Yaskawa INFORM job: DPRINT3D11.JBI

/JOB
//NAME DPRINT3D11
//POS
///NPOS 944,0,0,0,0,0
///TOOL 9
///POSTYPE PULSE
///PULSE
C00000=39305,52973,-116691,73872,-117726,-90951,0
C00001=43922,55434,-109343,70072,-122046,-89427,0
C00002=34855,54702,-111321,79150,-116923,-88842,0
C00003=33073,56542,-105908,81594,-117099,-87037,0
C00004=36075,53739,-114252,77543,-116850,-89855,0
C00005=40141,50956,-123257,72181,-116164,-93028,0
C00006=40141,50893,-123279,72189,-116185,-93006,0
C00007=25718,54883,-110483,67428,-122670,-90024,0
C00008=36367,51719,-120456,76529,-115448,-91749,0
C00009=36299,54106,-112987,77479,-117287,-89472,0
C00010=40952,50916,-123219,71325,-116516,-93076,0
C00011=39945,50531,-124504,72259,-115736,-93361,0
C00012=35336,53692,-114225,78320,-116517,-89741,0
C00013=36221,54071,-113090,77546,-117224,-89494,0
C00014=35607,54392,-112113,78297,-117147,-89134,0
C00015=36480,54789,-110943,77551,-117869,-88882,0
C00016=42179,50883,-123364,69985,-116939,-93256,0
C00017=33604,54402,-112044,58649,-125681,-91811,0
C00018=34235,53812,-113837,79497,-116065,-89510,0
C00019=35137,54187,-112719,78704,-116769,-89265,0
C00020=34902,54401,-112073,79022,-116798,-89046,0
C00021=35370,54606,-111468,78618,-117176,-88914,0
C00022=35553,54440,-111967,78370,-117154,-89084,0
C00023=36112,54158,-112826,77691,-117233,-89403,0
C00024=41179,50259,-125479,70816,-115885,-93789,0
C00025=36778,53010,-116357,54404,-125157,-93511,0
C00026=39305,52913,-116713,73881,-117747,-90930,0
C00027=43892,55358,-109419,70105,-122035,-89419,0
C00028=34855,54645,-111342,79158,-116939,-88821,0
C00029=33085,56473,-105968,81585,-117112,-87030,0
C00030=36076,53681,-114273,77551,-116867,-89834,0
C00031=40141,50893,-123279,72189,-116185,-93006,0
C00032=40142,50830,-123301,72197,-116208,-92984,0
C00033=25756,54837,-110470,67404,-122722,-90001,0
C00034=36367,51658,-120476,76537,-115466,-91727,0
C00035=36299,54048,-113008,77487,-117305,-89450,0
C00036=40952,50853,-123241,71333,-116539,-93053,0
C00037=39946,50468,-124526,72267,-115759,-93339,0
C00038=35336,53633,-114246,78328,-116535,-89719,0
C00039=36221,54013,-113111,77555,-117241,-89473,0
C00040=35607,54334,-112134,78305,-117163,-89113,0
C00041=36480,54732,-110963,77560,-117886,-88861,0
C00042=42180,50820,-123386,69993,-116962,-93234,0
C00043=33604,54344,-112065,58660,-125708,-91792,0
C00044=34236,53754,-113858,79505,-116081,-89488,0
C00045=35137,54129,-112740,78712,-116785,-89244,0
C00046=34902,54343,-112094,79030,-116814,-89025,0
C00047=35370,54548,-111489,78626,-117192,-88894,0
C00048=35553,54382,-111988,78379,-117170,-89063,0
C00049=36113,54100,-112847,77699,-117251,-89382,0
C00050=41180,50194,-125500,70824,-115910,-93766,0
C00051=36764,52962,-116343,54437,-125197,-93481,0
C00052=39305,52854,-116734,73889,-117767,-90909,0
C00053=43862,55283,-109495,70139,-122024,-89410,0
C00054=34856,54587,-111363,79166,-116954,-88801,0
C00055=33098,56404,-106029,81577,-117124,-87023,0
C00056=36076,53622,-114294,77560,-116884,-89813,0
C00057=40142,50830,-123301,72197,-116208,-92984,0
C00058=40142,50767,-123323,72205,-116231,-92961,0
C00059=25794,54792,-110456,67381,-122773,-89978,0
C00060=36368,51596,-120498,76545,-115486,-91704,0
C00061=36299,53990,-113029,77496,-117322,-89430,0
C00062=40952,50790,-123263,71342,-116562,-93031,0
C00063=39946,50404,-124548,72275,-115782,-93316,0
C00064=35337,53575,-114267,78336,-116551,-89698,0
C00065=36222,53955,-113131,77563,-117258,-89452,0
C00066=35607,54276,-112155,78314,-117179,-89092,0
C00067=36480,54675,-110984,77568,-117902,-88841,0
C00068=42180,50757,-123408,70002,-116986,-93212,0
C00069=33604,54287,-112086,58672,-125736,-91774,0
C00070=34236,53695,-113879,79512,-116097,-89467,0
C00071=35137,54071,-112761,78721,-116801,-89223,0
C00072=34902,54285,-112114,79038,-116830,-89004,0
C00073=35371,54491,-111509,78635,-117208,-88873,0
C00074=35553,54325,-112009,78387,-117186,-89042,0
C00075=36113,54042,-112867,77707,-117267,-89360,0
C00076=41180,50130,-125522,70832,-115933,-93744,0
C00077=36749,52914,-116328,54470,-125238,-93452,0
C00078=39306,52794,-116755,73898,-117787,-90887,0
C00079=43832,55207,-109571,70173,-122014,-89401,0
C00080=34856,54530,-111383,79174,-116970,-88780,0
C00081=33110,56335,-106089,81568,-117137,-87016,0
C00082=36076,53564,-114315,77568,-116901,-89791,0
C00083=40142,50767,-123323,72205,-116231,-92961,0
C00084=40143,50704,-123345,72213,-116253,-92939,0
C00085=25832,54747,-110443,67357,-122825,-89955,0
C00086=36368,51535,-120519,76552,-115505,-91682,0
C00087=36300,53932,-113049,77504,-117339,-89409,0
C00088=40953,50727,-123285,71350,-116585,-93009,0
C00089=39947,50340,-124570,72283,-115805,-93293,0
C00090=35337,53516,-114288,78344,-116568,-89676,0
C00091=36222,53897,-113152,77571,-117275,-89431,0
C00092=35608,54219,-112176,78322,-117197,-89071,0
C00093=36481,54618,-111005,77577,-117919,-88820,0
C00094=42181,50693,-123430,70010,-117010,-93190,0
C00095=33605,54229,-112107,58684,-125764,-91756,0
C00096=34236,53637,-113900,79520,-116113,-89445,0
C00097=35138,54013,-112781,78729,-116819,-89201,0
C00098=34903,54228,-112135,79047,-116846,-88983,0
C00099=35371,54434,-111530,78643,-117224,-88852,0
C00100=35554,54267,-112029,78395,-117202,-89021,0
C00101=36113,53984,-112888,77716,-117284,-89340,0
C00102=41181,50066,-125544,70840,-115957,-93721,0
C00103=36735,52866,-116314,54503,-125279,-93422,0
C00104=39306,52734,-116776,73907,-117807,-90866,0
C00105=43802,55132,-109647,70206,-122004,-89393,0
C00106=34856,54473,-111404,79182,-116986,-88759,0
C00107=33122,56266,-106149,81559,-117150,-87008,0
C00108=36077,53505,-114336,77576,-116919,-89770,0
C00109=40143,50704,-123345,72213,-116253,-92939,0
C00110=40143,50641,-123365,72222,-116276,-92916,0
C00111=25870,54702,-110429,67334,-122878,-89931,0
C00112=36368,51473,-120541,76560,-115523,-91660,0
C00113=36300,53874,-113070,77513,-117356,-89388,0
C00114=40953,50664,-123307,71359,-116609,-92987,0
C00115=39947,50276,-124591,72291,-115828,-93270,0
C00116=35337,53458,-114308,78353,-116585,-89655,0
C00117=36222,53839,-113173,77580,-117292,-89410,0
C00118=35608,54161,-112196,78330,-117213,-89050,0
C00119=36481,54561,-111025,77586,-117937,-88799,0
C00120=42181,50630,-123450,70019,-117035,-93168,0
C00121=33605,54172,-112127,58695,-125791,-91738,0
C00122=34237,53579,-113920,79528,-116129,-89424,0
C00123=35138,53956,-112802,78737,-116835,-89181,0
C00124=34903,54170,-112156,79055,-116862,-88961,0
C00125=35371,54376,-111551,78651,-117240,-88831,0
C00126=35554,54210,-112050,78403,-117220,-89000,0
C00127=36114,53926,-112909,77724,-117301,-89319,0
C00128=41181,50001,-125565,70849,-115981,-93698,0
C00129=36721,52817,-116299,54537,-125320,-93393,0
C00130=39307,52675,-116797,73916,-117828,-90844,0
C00131=43772,55056,-109723,70240,-121992,-89384,0
C00132=34857,54416,-111425,79190,-117002,-88737,0
C00133=33135,56197,-106209,81551,-117162,-87001,0
C00134=36077,53447,-114357,77584,-116936,-89749,0
C00135=40143,50641,-123365,72222,-116276,-92916,0
C00136=40143,50578,-123387,72230,-116299,-92894,0
C00137=25908,54657,-110415,67310,-122930,-89908,0
C00138=36369,51412,-120561,76568,-115543,-91637,0
C00139=36300,53816,-113091,77521,-117374,-89366,0
C00140=40954,50601,-123327,71367,-116632,-92964,0
C00141=39947,50213,-124613,72299,-115851,-93247,0
C00142=35338,53399,-114329,78361,-116601,-89634,0
C00143=36223,53781,-113194,77588,-117309,-89388,0
C00144=35608,54104,-112217,78339,-117230,-89029,0
C00145=36481,54504,-111046,77594,-117953,-88778,0
C00146=42182,50567,-123472,70028,-117059,-93146,0
C00147=33605,54114,-112148,58707,-125819,-91720,0
C00148=34237,53520,-113941,79536,-116145,-89402,0
C00149=35138,53898,-112823,78745,-116851,-89159,0
C00150=34903,54113,-112176,79063,-116878,-88940,0
C00151=35372,54319,-111571,78659,-117256,-88810,0
C00152=35554,54152,-112070,78412,-117236,-88979,0
C00153=36114,53869,-112929,77733,-117318,-89297,0
C00154=41181,49937,-125587,70857,-116005,-93675,0
C00155=36707,52769,-116285,54570,-125361,-93363,0
C00156=39307,52615,-116817,73925,-117847,-90823,0
C00157=43742,54980,-109798,70274,-121982,-89376,0
C00158=34857,54358,-111445,79198,-117019,-88716,0
C00159=33147,56128,-106269,81542,-117175,-86994,0
C00160=36077,53388,-114377,77593,-116953,-89727,0
C00161=40143,50578,-123387,72230,-116299,-92894,0
C00162=40144,50515,-123408,72238,-116321,-92871,0
C00163=25945,54612,-110401,67287,-122981,-89886,0
C00164=36369,51351,-120583,76576,-115563,-91614,0
C00165=36301,53758,-113111,77530,-117391,-89345,0
C00166=40954,50538,-123349,71375,-116655,-92942,0
C00167=39948,50149,-124634,72307,-115874,-93224,0
C00168=35338,53341,-114350,78369,-116619,-89612,0
C00169=36223,53723,-113214,77597,-117326,-89367,0
C00170=35608,54046,-112237,78347,-117246,-89008,0
C00171=36482,54447,-111066,77603,-117970,-88758,0
C00172=42182,50504,-123493,70036,-117083,-93124,0
C00173=33606,54057,-112168,58719,-125846,-91701,0
C00174=34237,53462,-113962,79544,-116161,-89381,0
C00175=35139,53840,-112843,78753,-116867,-89138,0
C00176=34904,54055,-112197,79071,-116894,-88919,0
C00177=35372,54262,-111592,78668,-117272,-88789,0
C00178=35555,54095,-112091,78420,-117252,-88958,0
C00179=36114,53811,-112950,77741,-117336,-89276,0
C00180=41182,49873,-125608,70865,-116029,-93652,0
C00181=36693,52721,-116270,54603,-125402,-93334,0
C00182=39307,52556,-116838,73933,-117868,-90801,0
C00183=43712,54905,-109874,70308,-121971,-89367,0
C00184=34857,54301,-111466,79207,-117033,-88696,0
C00185=33159,56059,-106328,81533,-117189,-86986,0
C00186=36078,53330,-114398,77601,-116970,-89706,0
C00187=40144,50515,-123408,72238,-116321,-92871,0
C00188=40144,50452,-123430,72246,-116344,-92848,0
C00189=25983,54568,-110386,67264,-123034,-89862,0
C00190=36370,51289,-120604,76584,-115581,-91592,0
C00191=36301,53700,-113132,77538,-117408,-89324,0
C00192=40954,50476,-123370,71384,-116678,-92919,0
C00193=39948,50085,-124656,72315,-115897,-93201,0
C00194=35338,53283,-114370,78377,-116636,-89590,0
C00195=36223,53665,-113234,77605,-117344,-89346,0
C00196=35609,53989,-112258,78355,-117262,-88987,0
C00197=36482,54390,-111087,77612,-117986,-88737,0
C00198=42182,50441,-123515,70045,-117107,-93101,0
C00199=33606,53999,-112189,58731,-125875,-91683,0
C00200=34238,53404,-113982,79552,-116177,-89359,0
C00201=35139,53782,-112864,78762,-116884,-89117,0
C00202=34904,53998,-112217,79079,-116910,-88898,0
C00203=35372,54205,-111612,78676,-117289,-88768,0
C00204=35555,54037,-112111,78429,-117269,-88937,0
C00205=36115,53753,-112970,77749,-117352,-89255,0
C00206=41182,49809,-125630,70873,-116054,-93630,0
C00207=36679,52673,-116255,54636,-125443,-93304,0
C00208=39308,52496,-116859,73942,-117887,-90780,0
C00209=43682,54829,-109949,70342,-121960,-89358,0
C00210=34858,54244,-111486,79215,-117050,-88675,0
C00211=33172,55990,-106388,81524,-117201,-86979,0
C00212=36078,53271,-114418,77609,-116987,-89684,0
C00213=40144,50452,-123430,72246,-116344,-92848,0
C00214=40145,50389,-123450,72255,-116367,-92826,0
C00215=26021,54523,-110372,67241,-123086,-89839,0
C00216=36370,51228,-120625,76591,-115600,-91569,0
C00217=36302,53642,-113152,77547,-117425,-89302,0
C00218=40955,50413,-123391,71392,-116702,-92897,0
C00219=39949,50022,-124676,72323,-115920,-93179,0
C00220=35339,53224,-114391,78385,-116652,-89569,0
C00221=36224,53608,-113255,77614,-117361,-89325,0
C00222=35609,53931,-112278,78364,-117279,-88965,0
C00223=36482,54333,-111107,77621,-118003,-88716,0
C00224=42183,50378,-123535,70054,-117132,-93079,0
C00225=33606,53942,-112209,58743,-125903,-91665,0
C00226=34238,53346,-114003,79560,-116193,-89338,0
C00227=35139,53724,-112884,78770,-116900,-89095,0
C00228=34904,53940,-112238,79087,-116927,-88877,0
C00229=35373,54147,-111632,78685,-117306,-88747,0
C00230=35555,53980,-112132,78437,-117285,-88916,0
C00231=36115,53695,-112991,77758,-117369,-89234,0
C00232=41183,49744,-125651,70881,-116079,-93606,0
C00233=36665,52626,-116242,54670,-125483,-93274,0
C00234=39308,52436,-116879,73951,-117908,-90758,0
C00235=43651,54754,-110024,70376,-121950,-89349,0
C00236=34858,54187,-111506,79223,-117066,-88653,0
C00237=33184,55921,-106448,81516,-117214,-86972,0
C00238=36078,53213,-114439,77618,-117006,-89663,0
C00239=40145,50389,-123450,72255,-116367,-92826,0
C00240=40145,50326,-123471,72263,-116390,-92803,0
C00241=26059,54478,-110357,67218,-123139,-89816,0
C00242=36370,51166,-120645,76599,-115620,-91546,0
C00243=36302,53584,-113172,77555,-117443,-89282,0
C00244=40955,50350,-123412,71401,-116725,-92874,0
C00245=39949,49958,-124698,72331,-115943,-93155,0
C00246=35339,53166,-114411,78393,-116669,-89547,0
C00247=36224,53550,-113275,77622,-117378,-89304,0
C00248=35609,53874,-112298,78372,-117295,-88944,0
C00249=36483,54276,-111127,77629,-118021,-88695,0
C00250=42183,50315,-123556,70062,-117156,-93056,0
C00251=33607,53884,-112229,58755,-125930,-91646,0
C00252=34238,53288,-114023,79568,-116210,-89316,0
C00253=35140,53667,-112904,78778,-116916,-89074,0
C00254=34905,53883,-112258,79096,-116943,-88856,0
C00255=35373,54090,-111653,78693,-117322,-88726,0
C00256=35556,53923,-112152,78445,-117301,-88895,0
C00257=36115,53637,-113011,77766,-117386,-89213,0
C00258=41183,49680,-125673,70890,-116103,-93584,0
C00259=36650,52578,-116227,54703,-125525,-93245,0
C00260=39308,52377,-116900,73960,-117929,-90737,0
C00261=43621,54678,-110099,70410,-121939,-89340,0
C00262=34858,54130,-111527,79232,-117082,-88632,0
C00263=33197,55852,-106507,81507,-117227,-86964,0
C00264=36079,53155,-114459,77626,-117023,-89641,0
C00265=40145,50326,-123471,72263,-116390,-92803,0
C00266=40145,50263,-123493,72271,-116413,-92781,0
C00267=26097,54434,-110343,67195,-123191,-89793,0
C00268=36371,51105,-120666,76607,-115638,-91524,0
C00269=36302,53527,-113193,77564,-117460,-89260,0
C00270=40956,50287,-123433,71409,-116748,-92851,0
C00271=39949,49894,-124719,72339,-115966,-93133,0
C00272=35339,53107,-114431,78402,-116686,-89526,0
C00273=36224,53492,-113295,77631,-117395,-89282,0
C00274=35610,53816,-112318,78381,-117313,-88923,0
C00275=36483,54219,-111147,77638,-118038,-88674,0
C00276=42184,50252,-123578,70071,-117181,-93034,0
C00277=33607,53827,-112249,58767,-125959,-91628,0
C00278=34239,53229,-114043,79575,-116226,-89294,0
C00279=35140,53609,-112925,78786,-116933,-89053,0
C00280=34905,53825,-112278,79104,-116959,-88834,0
C00281=35373,54033,-111673,78702,-117338,-88705,0
C00282=35556,53865,-112172,78454,-117318,-88874,0
C00283=36116,53580,-113031,77775,-117403,-89192,0
C00284=41184,49616,-125693,70898,-116127,-93560,0
C00285=36636,52530,-116212,54736,-125565,-93215,0
C00286=39309,52317,-116921,73969,-117948,-90715,0
C00287=43591,54602,-110174,70444,-121929,-89331,0
C00288=34859,54073,-111547,79240,-117098,-88611,0
C00289=33209,55783,-106566,81498,-117240,-86956,0
C00290=36079,53096,-114480,77635,-117040,-89620,0
C00291=40145,50263,-123493,72271,-116413,-92781,0
C00292=40146,50200,-123514,72280,-116436,-92757,0
C00293=26135,54389,-110328,67172,-123243,-89770,0
C00294=36371,51043,-120687,76615,-115658,-91501,0
C00295=36303,53469,-113213,77572,-117477,-89239,0
C00296=40956,50224,-123454,71418,-116773,-92829,0
C00297=39950,49831,-124740,72348,-115989,-93110,0
C00298=35340,53049,-114451,78410,-116704,-89504,0
C00299=36225,53434,-113315,77639,-117413,-89261,0
C00300=35610,53759,-112338,78389,-117329,-88901,0
C00301=36483,54162,-111167,77647,-118054,-88653,0
C00302=42184,50189,-123599,70080,-117205,-93012,0
C00303=33607,53769,-112269,58779,-125987,-91610,0
C00304=34239,53171,-114063,79584,-116242,-89273,0
C00305=35140,53551,-112945,78795,-116950,-89031,0
C00306=34905,53768,-112298,79112,-116975,-88813,0
C00307=35374,53976,-111693,78710,-117354,-88683,0
C00308=35556,53808,-112192,78462,-117335,-88852,0
C00309=36116,53522,-113051,77784,-117421,-89170,0
C00310=41184,49552,-125714,70906,-116151,-93537,0
C00311=36622,52482,-116196,54770,-125606,-93185,0
C00312=39309,52258,-116940,73978,-117969,-90694,0
C00313=43561,54527,-110249,70478,-121919,-89322,0
C00314=34859,54015,-111567,79248,-117114,-88590,0
C00315=33222,55714,-106626,81490,-117253,-86949,0
C00316=36079,53038,-114500,77643,-117058,-89598,0
C00317=40146,50200,-123514,72280,-116436,-92757,0
C00318=40146,50137,-123534,72288,-116458,-92735,0
C00319=26173,54345,-110313,67149,-123295,-89746,0
C00320=36371,50982,-120707,76623,-115677,-91478,0
C00321=36303,53411,-113233,77581,-117494,-89218,0
C00322=40956,50161,-123474,71427,-116796,-92806,0
C00323=39950,49767,-124762,72356,-116012,-93086,0
C00324=35340,52991,-114472,78418,-116720,-89482,0
C00325=36225,53376,-113336,77648,-117430,-89239,0
C00326=35611,53701,-112358,78398,-117346,-88881,0
C00327=36484,54105,-111187,77656,-118071,-88632,0
C00328=42184,50126,-123619,70089,-117229,-92989,0
C00329=33608,53712,-112289,58790,-126014,-91591,0
C00330=34239,53113,-114083,79591,-116258,-89251,0
C00331=35141,53494,-112965,78803,-116966,-89010,0
C00332=34906,53710,-112318,79121,-116991,-88792,0
C00333=35374,53919,-111713,78718,-117370,-88662,0
C00334=35556,53750,-112212,78471,-117352,-88831,0
C00335=36116,53464,-113071,77792,-117438,-89149,0
C00336=41184,49487,-125736,70915,-116175,-93515,0
C00337=36608,52435,-116181,54804,-125646,-93155,0
C00338=39310,52199,-116961,73987,-117988,-90672,0
C00339=43530,54451,-110324,70512,-121908,-89313,0
C00340=34859,53958,-111587,79257,-117130,-88569,0
C00341=33234,55645,-106685,81481,-117267,-86941,0
C00342=36080,52979,-114520,77652,-117075,-89576,0
C00343=40146,50137,-123534,72288,-116458,-92735,0
C00344=40147,50074,-123555,72297,-116481,-92712,0
C00345=26210,54300,-110298,67126,-123348,-89723,0
C00346=36372,50921,-120728,76631,-115697,-91455,0
C00347=36303,53353,-113253,77590,-117511,-89196,0
C00348=40957,50098,-123495,71435,-116819,-92783,0
C00349=39951,49704,-124782,72364,-116035,-93063,0
C00350=35340,52932,-114492,78427,-116737,-89461,0
C00351=36225,53318,-113355,77657,-117447,-89218,0
C00352=35611,53644,-112378,78406,-117362,-88859,0
C00353=36484,54048,-111207,77665,-118088,-88611,0
C00354=42185,50063,-123640,70098,-117253,-92967,0
C00355=33608,53655,-112309,58803,-126043,-91572,0
C00356=34239,53055,-114103,79599,-116274,-89229,0
C00357=35141,53436,-112985,78811,-116983,-88989,0
C00358=34906,53653,-112338,79129,-117007,-88770,0
C00359=35374,53862,-111733,78727,-117387,-88641,0
C00360=35557,53693,-112232,78480,-117368,-88810,0
C00361=36117,53406,-113091,77801,-117455,-89127,0
C00362=41185,49423,-125757,70923,-116199,-93491,0
C00363=36594,52387,-116166,54837,-125688,-93126,0
C00364=39310,52139,-116981,73996,-118009,-90650,0
C00365=43500,54376,-110398,70546,-121898,-89304,0
C00366=34860,53901,-111607,79265,-117146,-88548,0
C00367=33247,55577,-106744,81473,-117279,-86934,0
C00368=36080,52921,-114540,77660,-117093,-89555,0
C00369=40147,50074,-123555,72297,-116481,-92712,0
C00370=40147,50011,-123576,72305,-116504,-92689,0
C00371=26248,54256,-110282,67104,-123401,-89700,0
C00372=36372,50859,-120748,76639,-115717,-91433,0
C00373=36304,53296,-113273,77598,-117529,-89175,0
C00374=40957,50035,-123516,71444,-116843,-92761,0
C00375=39951,49640,-124803,72372,-116058,-93040,0
C00376=35341,52874,-114512,78435,-116754,-89439,0
C00377=36226,53260,-113375,77665,-117464,-89196,0
C00378=35611,53587,-112398,78415,-117379,-88838,0
C00379=36484,53991,-111227,77674,-118106,-88590,0
C00380=42185,50000,-123661,70106,-117278,-92944,0
C00381=33608,53597,-112329,58815,-126070,-91554,0
C00382=34240,52997,-114123,79608,-116290,-89207,0
C00383=35141,53378,-113004,78820,-116999,-88967,0
C00384=34906,53596,-112358,79137,-117023,-88749,0
C00385=35375,53805,-111753,78736,-117403,-88620,0
C00386=35557,53636,-112252,78488,-117385,-88788,0
C00387=36117,53349,-113111,77809,-117472,-89106,0
C00388=41185,49359,-125777,70931,-116224,-93468,0
C00389=36580,52340,-116151,54871,-125728,-93096,0
C00390=39310,52080,-117001,74006,-118030,-90628,0
C00391=43470,54300,-110472,70580,-121887,-89295,0
C00392=34860,53844,-111626,79273,-117162,-88526,0
C00393=33259,55508,-106803,81464,-117292,-86926,0
C00394=36080,52863,-114560,77669,-117110,-89533,0
C00395=40147,50011,-123576,72305,-116504,-92689,0
C00396=40147,49948,-123596,72314,-116527,-92666,0
C00397=26286,54212,-110267,67081,-123454,-89677,0
C00398=36372,50798,-120768,76647,-115736,-91409,0
C00399=36304,53238,-113292,77607,-117546,-89153,0
C00400=40958,49973,-123537,71453,-116866,-92738,0
C00401=39951,49576,-124824,72381,-116081,-93017,0
C00402=35341,52816,-114531,78443,-116771,-89417,0
C00403=36226,53203,-113395,77674,-117482,-89175,0
C00404=35611,53529,-112418,78424,-117395,-88816,0
C00405=36485,53934,-111247,77682,-118122,-88569,0
C00406=42186,49938,-123681,70115,-117302,-92922,0
C00407=33608,53540,-112349,58827,-126098,-91535,0
C00408=34240,52939,-114143,79616,-116306,-89186,0
C00409=35142,53321,-113024,78828,-117016,-88946,0
C00410=34907,53538,-112378,79146,-117039,-88727,0
C00411=35375,53747,-111772,78744,-117420,-88599,0
C00412=35557,53579,-112272,78497,-117401,-88767,0
C00413=36117,53291,-113131,77818,-117490,-89084,0
C00414=41186,49295,-125798,70940,-116249,-93445,0
C00415=36566,52292,-116135,54904,-125769,-93066,0
C00416=39311,52020,-117021,74015,-118050,-90607,0
C00417=43439,54224,-110547,70615,-121877,-89286,0
C00418=34860,53787,-111646,79282,-117178,-88505,0
C00419=33272,55439,-106862,81455,-117306,-86918,0
C00420=36081,52805,-114580,77677,-117128,-89511,0
C00421=40147,49948,-123596,72314,-116527,-92666,0
C00422=40148,49886,-123617,72322,-116550,-92643,0
C00423=26324,54168,-110251,67059,-123507,-89654,0
C00424=36373,50737,-120788,76655,-115754,-91387,0
C00425=36304,53180,-113312,77616,-117563,-89132,0
C00426=40958,49910,-123557,71461,-116890,-92715,0
C00427=39952,49513,-124844,72389,-116105,-92994,0
C00428=35341,52758,-114551,78452,-116789,-89395,0
C00429=36226,53145,-113415,77683,-117500,-89153,0
C00430=35612,53472,-112438,78432,-117413,-88795,0
C00431=36485,53877,-111266,77691,-118139,-88548,0
C00432=42186,49875,-123702,70124,-117326,-92899,0
C00433=33609,53483,-112369,58839,-126127,-91517,0
C00434=34241,52881,-114163,79624,-116322,-89164,0
C00435=35142,53263,-113044,78837,-117032,-88924,0
C00436=34907,53481,-112397,79154,-117056,-88706,0
C00437=35375,53690,-111792,78753,-117436,-88577,0
C00438=35558,53521,-112291,78505,-117418,-88745,0
C00439=36118,53233,-113151,77827,-117507,-89063,0
C00440=41186,49231,-125819,70948,-116273,-93422,0
C00441=36552,52245,-116120,54938,-125810,-93036,0
C00442=39311,51961,-117041,74024,-118070,-90585,0
C00443=43409,54149,-110621,70649,-121867,-89276,0
C00444=34861,53730,-111666,79290,-117194,-88484,0
C00445=33284,55370,-106921,81447,-117320,-86911,0
C00446=36081,52746,-114599,77686,-117145,-89490,0
C00447=40148,49886,-123617,72322,-116550,-92643,0
C00448=40148,49823,-123636,72331,-116573,-92620,0
C00449=26361,54124,-110236,67037,-123560,-89630,0
C00450=36373,50676,-120808,76663,-115774,-91364,0
C00451=36304,53122,-113332,77625,-117580,-89110,0
C00452=40958,49847,-123577,71470,-116913,-92692,0
C00453=39952,49449,-124864,72398,-116128,-92970,0
C00454=35342,52699,-114571,78460,-116805,-89374,0
C00455=36227,53087,-113435,77692,-117517,-89132,0
C00456=35612,53415,-112457,78441,-117429,-88774,0
C00457=36485,53821,-111286,77700,-118156,-88527,0
C00458=42187,49812,-123722,70133,-117351,-92876,0
C00459=33609,53425,-112388,58851,-126154,-91498,0
C00460=34241,52823,-114183,79632,-116338,-89142,0
C00461=35142,53206,-113064,78845,-117048,-88903,0
C00462=34907,53424,-112417,79163,-117073,-88684,0
C00463=35376,53633,-111811,78761,-117453,-88556,0
C00464=35558,53464,-112311,78514,-117435,-88725,0
C00465=36118,53176,-113170,77836,-117524,-89041,0
C00466=41187,49167,-125839,70957,-116298,-93399,0
C00467=36538,52197,-116104,54972,-125850,-93006,0
C00468=39311,51901,-117061,74033,-118091,-90563,0
C00469=43378,54073,-110695,70684,-121856,-89267,0
C00470=34861,53673,-111685,79299,-117210,-88462,0
C00471=33296,55301,-106979,81438,-117332,-86902,0
C00472=36081,52688,-114619,77694,-117163,-89468,0
C00473=40148,49823,-123636,72331,-116573,-92620,0
C00474=40149,49760,-123657,72340,-116596,-92597,0
C00475=26399,54080,-110220,67014,-123612,-89607,0
C00476=36374,50614,-120828,76672,-115794,-91341,0
C00477=36305,53065,-113351,77633,-117598,-89089,0
C00478=40959,49784,-123597,71479,-116937,-92670,0
C00479=39953,49386,-124884,72406,-116151,-92947,0
C00480=35342,52641,-114590,78468,-116822,-89352,0
C00481=36227,53029,-113454,77700,-117534,-89110,0
C00482=35612,53357,-112477,78449,-117446,-88752,0
C00483=36486,53764,-111305,77709,-118173,-88506,0
C00484=42187,49749,-123742,70142,-117376,-92854,0
C00485=33609,53368,-112408,58863,-126183,-91480,0
C00486=34241,52764,-114202,79640,-116354,-89120,0
C00487=35143,53148,-113083,78853,-117066,-88881,0
C00488=34908,53366,-112436,79171,-117089,-88663,0
C00489=35376,53576,-111831,78770,-117469,-88535,0
C00490=35558,53407,-112330,78522,-117452,-88703,0
C00491=36118,53118,-113190,77844,-117541,-89020,0
C00492=41187,49103,-125860,70965,-116322,-93375,0
C00493=36524,52150,-116089,55005,-125891,-92976,0
C00494=39312,51842,-117081,74042,-118111,-90541,0
C00495=43348,53998,-110769,70718,-121846,-89258,0
C00496=34861,53616,-111705,79307,-117227,-88441,0
C00497=33309,55232,-107038,81430,-117346,-86895,0
C00498=36082,52630,-114639,77703,-117181,-89446,0
C00499=40149,49760,-123657,72340,-116596,-92597,0
C00500=40149,49697,-123677,72348,-116619,-92574,0
C00501=26437,54036,-110204,66992,-123665,-89584,0
C00502=36374,50553,-120849,76680,-115813,-91318,0
C00503=36305,53007,-113371,77642,-117616,-89067,0
C00504=40959,49721,-123618,71488,-116960,-92647,0
C00505=39953,49322,-124905,72414,-116174,-92924,0
C00506=35342,52583,-114610,78477,-116839,-89330,0
C00507=36227,52972,-113474,77709,-117552,-89089,0
C00508=35613,53300,-112496,78458,-117463,-88731,0
C00509=36486,53707,-111325,77718,-118191,-88484,0
C00510=42187,49686,-123763,70151,-117400,-92831,0
C00511=33610,53311,-112427,58875,-126211,-91460,0
C00512=34241,52706,-114222,79648,-116372,-89098,0
C00513=35143,53091,-113103,78862,-117082,-88859,0
C00514=34908,53309,-112456,79179,-117105,-88642,0
C00515=35376,53519,-111850,78779,-117485,-88513,0
C00516=35559,53350,-112350,78531,-117468,-88682,0
C00517=36119,53061,-113209,77853,-117559,-88998,0
C00518=41187,49038,-125881,70974,-116346,-93352,0
C00519=36510,52103,-116073,55039,-125931,-92946,0
C00520=39312,51783,-117100,74051,-118132,-90519,0
C00521=43318,53922,-110842,70753,-121836,-89248,0
C00522=34861,53559,-111724,79316,-117243,-88419,0
C00523=33322,55163,-107097,81421,-117359,-86887,0
C00524=36082,52571,-114658,77712,-117198,-89424,0
C00525=40149,49697,-123677,72348,-116619,-92574,0
C00526=40149,49634,-123697,72357,-116642,-92551,0
C00527=26474,53992,-110188,66970,-123718,-89561,0
C00528=36374,50492,-120868,76688,-115833,-91295,0
C00529=36306,52950,-113390,77651,-117633,-89045,0
C00530=40960,49659,-123638,71497,-116984,-92624,0
C00531=39954,49259,-124925,72423,-116198,-92901,0
C00532=35343,52525,-114629,78485,-116856,-89308,0
C00533=36228,52914,-113493,77718,-117569,-89067,0
C00534=35613,53243,-112516,78467,-117479,-88709,0
C00535=36486,53650,-111344,77727,-118207,-88463,0
C00536=42188,49623,-123782,70160,-117425,-92808,0
C00537=33610,53254,-112446,58888,-126239,-91442,0
C00538=34242,52648,-114241,79656,-116388,-89076,0
C00539=35143,53033,-113122,78871,-117099,-88838,0
C00540=34908,53252,-112475,79188,-117121,-88620,0
C00541=35377,53462,-111870,78787,-117502,-88492,0
C00542=35559,53292,-112369,78540,-117485,-88660,0
C00543=36119,53003,-113229,77862,-117576,-88977,0
C00544=41188,48974,-125900,70982,-116372,-93328,0
C00545=36496,52056,-116057,55073,-125973,-92916,0
C00546=39312,51723,-117120,74061,-118152,-90498,0
C00547=43287,53847,-110916,70787,-121827,-89239,0
C00548=34862,53502,-111744,79324,-117259,-88398,0
C00549=33334,55094,-107155,81413,-117372,-86879,0
C00550=36082,52513,-114678,77720,-117216,-89403,0
C00551=40149,49634,-123697,72357,-116642,-92551,0
C00552=40150,49572,-123717,72366,-116665,-92528,0
C00553=26512,53948,-110172,66948,-123771,-89537,0
C00554=36375,50431,-120888,76696,-115852,-91272,0
C00555=36306,52892,-113409,77660,-117651,-89024,0
C00556=40960,49596,-123658,71506,-117007,-92601,0
C00557=39954,49195,-124945,72432,-116221,-92877,0
C00558=35343,52467,-114649,78494,-116874,-89286,0
C00559=36228,52856,-113512,77727,-117586,-89045,0
C00560=35613,53185,-112535,78475,-117497,-88687,0
C00561=36487,53593,-111363,77736,-118224,-88442,0
C00562=42188,49560,-123802,70170,-117449,-92785,0
C00563=33610,53196,-112466,58900,-126268,-91423,0
C00564=34242,52590,-114260,79665,-116404,-89054,0
C00565=35144,52976,-113141,78879,-117115,-88816,0
C00566=34909,53195,-112494,79197,-117137,-88599,0
C00567=35377,53405,-111889,78796,-117518,-88470,0
C00568=35559,53235,-112388,78549,-117501,-88638,0
C00569=36119,52946,-113248,77871,-117593,-88955,0
C00570=41188,48910,-125921,70991,-116396,-93305,0
C00571=36482,52008,-116041,55107,-126013,-92886,0
C00572=39313,51664,-117139,74070,-118172,-90476,0
C00573=43257,53771,-110990,70822,-121816,-89229,0
C00574=34862,53445,-111763,79333,-117275,-88376,0
C00575=33347,55025,-107213,81404,-117386,-86871,0
C00576=36083,52455,-114697,77729,-117233,-89381,0
C00577=40150,49572,-123717,72366,-116665,-92528,0
C00578=40150,49509,-123738,72375,-116688,-92505,0
C00579=26549,53905,-110155,66926,-123824,-89514,0
C00580=36375,50369,-120907,76704,-115872,-91249,0
C00581=36306,52834,-113429,77669,-117668,-89002,0
C00582=40961,49533,-123678,71514,-117031,-92578,0
C00583=39954,49132,-124965,72440,-116244,-92854,0
C00584=35343,52408,-114668,78502,-116891,-89264,0
C00585=36228,52799,-113532,77735,-117603,-89024,0
C00586=35614,53128,-112554,78484,-117513,-88666,0
C00587=36487,53537,-111382,77746,-118241,-88420,0
C00588=42189,49498,-123823,70179,-117474,-92763,0
C00589=33611,53139,-112485,58912,-126296,-91404,0
C00590=34242,52532,-114280,79673,-116420,-89032,0
C00591=35144,52918,-113160,78888,-117132,-88794,0
C00592=34909,53138,-112514,79205,-117154,-88577,0
C00593=35377,53348,-111908,78805,-117536,-88449,0
C00594=35560,53178,-112408,78557,-117518,-88617,0
C00595=36120,52888,-113267,77880,-117610,-88933,0
C00596=41189,48846,-125942,71000,-116420,-93282,0
C00597=36468,51961,-116024,55141,-126053,-92855,0
C00598=39313,51605,-117159,74079,-118193,-90454,0
C00599=43226,53695,-111063,70857,-121806,-89219,0
C00600=34862,53388,-111782,79341,-117291,-88355,0
C00601=33359,54956,-107271,81396,-117400,-86863,0
C00602=36083,52397,-114716,77738,-117251,-89359,0
C00603=40150,49509,-123738,72375,-116688,-92505,0
C00604=40151,49446,-123757,72383,-116712,-92482,0
C00605=26587,53861,-110139,66905,-123878,-89490,0
C00606=36375,50308,-120927,76713,-115891,-91225,0
C00607=36307,52777,-113448,77678,-117685,-88980,0
C00608=40961,49470,-123697,71523,-117055,-92555,0
C00609=39955,49068,-124986,72449,-116268,-92830,0
C00610=35344,52350,-114687,78511,-116908,-89242,0
C00611=36229,52741,-113551,77744,-117622,-89002,0
C00612=35614,53071,-112573,78493,-117530,-88644,0
C00613=36487,53480,-111402,77755,-118258,-88399,0
C00614=42189,49435,-123842,70188,-117499,-92740,0
C00615=33611,53082,-112504,58925,-126324,-91386,0
C00616=34243,52474,-114299,79681,-116436,-89010,0
C00617=35144,52861,-113180,78896,-117148,-88772,0
C00618=34909,53080,-112533,79214,-117170,-88555,0
C00619=35378,53291,-111927,78813,-117552,-88427,0
C00620=35560,53121,-112427,78566,-117534,-88595,0
C00621=36120,52830,-113286,77888,-117628,-88912,0
C00622=41189,48782,-125961,71008,-116445,-93258,0
C00623=36454,51914,-116008,55175,-126095,-92825,0
C00624=39314,51545,-117178,74088,-118214,-90432,0
C00625=43195,53620,-111136,70892,-121796,-89209,0
C00626=34863,53332,-111801,79350,-117307,-88333,0
C00627=33372,54887,-107330,81388,-117413,-86855,0
C00628=36083,52339,-114736,77746,-117269,-89337,0
C00629=40151,49446,-123757,72383,-116712,-92482,0
C00630=40151,49383,-123777,72392,-116735,-92459,0
C00631=26624,53817,-110122,66883,-123931,-89467,0
C00632=36376,50247,-120946,76721,-115911,-91202,0
C00633=36307,52719,-113467,77686,-117703,-88959,0
C00634=40961,49408,-123717,71532,-117078,-92532,0
C00635=39955,49005,-125005,72457,-116291,-92807,0
C00636=35344,52292,-114706,78519,-116925,-89220,0
C00637=36229,52684,-113570,77753,-117639,-88980,0
C00638=35614,53014,-112592,78502,-117547,-88623,0
C00639=36488,53423,-111421,77764,-118276,-88378,0
C00640=42190,49372,-123862,70197,-117523,-92717,0
C00641=33611,53025,-112523,58937,-126353,-91367,0
C00642=34243,52417,-114318,79689,-116453,-88988,0
C00643=35145,52803,-113199,78905,-117166,-88751,0
C00644=34909,53023,-112552,79222,-117186,-88534,0
C00645=35378,53235,-111946,78822,-117568,-88406,0
C00646=35560,53064,-112446,78575,-117552,-88574,0
C00647=36120,52773,-113305,77897,-117645,-88890,0
C00648=41190,48718,-125981,71017,-116469,-93235,0
C00649=36440,51867,-115991,55209,-126135,-92795,0
C00650=39314,51486,-117198,74098,-118234,-90410,0
C00651=43165,53544,-111209,70926,-121786,-89200,0
C00652=34863,53275,-111820,79359,-117323,-88312,0
C00653=33384,54818,-107388,81379,-117426,-86847,0
C00654=36084,52281,-114755,77755,-117286,-89315,0
C00655=40151,49383,-123777,72392,-116735,-92459,0
C00656=40151,49321,-123796,72401,-116758,-92435,0
C00657=26662,53774,-110105,66861,-123984,-89443,0
C00658=36376,50186,-120966,76729,-115930,-91179,0
C00659=36307,52662,-113486,77695,-117721,-88937,0
C00660=40962,49345,-123738,71541,-117102,-92508,0
C00661=39956,48941,-125025,72466,-116314,-92783,0
C00662=35344,52234,-114725,78528,-116943,-89198,0
C00663=36229,52626,-113589,77762,-117656,-88958,0
C00664=35615,52957,-112611,78511,-117563,-88601,0
C00665=36488,53367,-111439,77773,-118293,-88357,0
C00666=42190,49309,-123882,70206,-117548,-92694,0
C00667=33612,52968,-112542,58950,-126381,-91348,0
C00668=34243,52359,-114337,79698,-116469,-88966,0
C00669=35145,52746,-113218,78914,-117182,-88729,0
C00670=34910,52966,-112571,79231,-117202,-88512,0
C00671=35378,53178,-111965,78831,-117585,-88384,0
C00672=35561,53007,-112465,78584,-117569,-88552,0
C00673=36121,52716,-113324,77906,-117662,-88868,0
C00674=41190,48654,-126001,71026,-116494,-93211,0
C00675=36426,51821,-115975,55243,-126175,-92765,0
C00676=39314,51427,-117216,74107,-118255,-90388,0
C00677=43134,53469,-111282,70961,-121776,-89190,0
C00678=34863,53218,-111839,79367,-117339,-88290,0
C00679=33397,54749,-107445,81371,-117440,-86839,0
C00680=36084,52223,-114774,77764,-117305,-89293,0
C00681=40151,49321,-123796,72401,-116758,-92435,0
C00682=40152,49258,-123816,72410,-116781,-92412,0
C00683=26699,53731,-110088,66840,-124038,-89420,0
C00684=36376,50125,-120985,76738,-115950,-91156,0
C00685=36308,52604,-113505,77704,-117738,-88915,0
C00686=40962,49282,-123757,71550,-117127,-92486,0
C00687=39956,48878,-125045,72474,-116338,-92760,0
C00688=35344,52176,-114744,78537,-116960,-89175,0
C00689=36230,52568,-113608,77771,-117674,-88937,0
C00690=35615,52900,-112630,78520,-117580,-88579,0
C00691=36488,53310,-111458,77782,-118310,-88335,0
C00692=42190,49246,-123902,70215,-117572,-92671,0
C00693=39823,48305,-126937,72401,-115720,-93319,0
C00694=34244,52301,-114356,79706,-116485,-88944,0
C00695=35145,52688,-113237,78922,-117199,-88707,0
C00696=34910,52909,-112590,79240,-117220,-88490,0
C00697=35378,53121,-111984,78840,-117601,-88362,0
C00698=35561,52950,-112484,78593,-117585,-88530,0
C00699=36121,52658,-113343,77915,-117680,-88846,0
C00700=41190,48590,-126021,71034,-116519,-93188,0
C00701=36412,51774,-115959,55277,-126216,-92735,0
C00702=39315,51368,-117236,74117,-118275,-90366,0
C00703=43103,53393,-111355,70996,-121766,-89179,0
C00704=34864,53161,-111858,79376,-117355,-88268,0
C00705=33409,54680,-107503,81362,-117454,-86831,0
C00706=36084,52165,-114793,77773,-117322,-89271,0
C00707=40152,49258,-123816,72410,-116781,-92412,0
C00708=40152,49195,-123835,72419,-116804,-92389,0
C00709=26737,53687,-110071,66818,-124090,-89397,0
C00710=36377,50064,-121005,76746,-115969,-91133,0
C00711=36308,52547,-113524,77713,-117756,-88893,0
C00712=40963,49220,-123777,71559,-117150,-92463,0
C00713=39956,48814,-125065,72483,-116361,-92736,0
C00714=35345,52118,-114763,78545,-116977,-89153,0
C00715=36230,52511,-113626,77780,-117692,-88915,0
C00716=35615,52842,-112649,78528,-117598,-88558,0
C00717=36489,53253,-111477,77791,-118327,-88314,0
C00718=42191,49184,-123921,70225,-117598,-92648,0
C00719=39823,48241,-126956,72410,-115744,-93295,0
C00720=34244,52243,-114375,79714,-116501,-88922,0
C00721=35146,52631,-113255,78931,-117215,-88685,0
C00722=34911,52852,-112608,79248,-117236,-88468,0
C00723=35379,53064,-112003,78849,-117618,-88341,0
C00724=35561,52893,-112502,78601,-117602,-88509,0
C00725=36121,52601,-113362,77924,-117698,-88825,0
C00726=41191,48526,-126041,71043,-116544,-93164,0
C00727=36398,51727,-115942,55311,-126257,-92705,0
C00728=39315,51308,-117255,74126,-118295,-90343,0
C00729=43073,53318,-111428,71031,-121756,-89170,0
C00730=34864,53104,-111877,79385,-117371,-88247,0
C00731=33422,54611,-107561,81354,-117468,-86822,0
C00732=36085,52106,-114812,77782,-117339,-89248,0
C00733=40152,49195,-123835,72419,-116804,-92389,0
C00734=40153,49133,-123855,72428,-116828,-92366,0
C00735=26774,53644,-110054,66797,-124144,-89373,0
C00736=36377,50003,-121024,76754,-115989,-91109,0
C00737=36308,52489,-113542,77722,-117774,-88872,0
C00738=40963,49157,-123796,71568,-117174,-92439,0
C00739=39957,48751,-125084,72492,-116385,-92713,0
C00740=35345,52060,-114782,78554,-116994,-89131,0
C00741=36230,52453,-113645,77789,-117709,-88893,0
C00742=35616,52785,-112667,78537,-117615,-88536,0
C00743=36489,53197,-111496,77801,-118345,-88292,0
C00744=42191,49121,-123941,70234,-117622,-92625,0
C00745=39824,48176,-126977,72418,-115768,-93271,0
C00746=34244,52185,-114394,79723,-116519,-88899,0
C00747=35146,52574,-113274,78940,-117232,-88663,0
C00748=34911,52795,-112627,79257,-117252,-88446,0
C00749=35379,53007,-112021,78858,-117634,-88319,0
C00750=35562,52836,-112521,78610,-117620,-88487,0
C00751=36122,52543,-113381,77933,-117715,-88803,0
C00752=41191,48462,-126060,71052,-116568,-93140,0
C00753=36384,51680,-115926,55345,-126297,-92674,0
C00754=39315,51249,-117274,74136,-118316,-90321,0
C00755=43042,53242,-111500,71066,-121746,-89160,0
C00756=34864,53048,-111895,79394,-117387,-88225,0
C00757=33434,54543,-107619,81346,-117482,-86814,0
C00758=36085,52048,-114830,77790,-117358,-89226,0
C00759=40153,49133,-123855,72428,-116828,-92366,0
C00760=40153,49070,-123874,72437,-116851,-92342,0
C00761=26811,53601,-110037,66776,-124198,-89350,0
C00762=36377,49941,-121043,76763,-116008,-91086,0
C00763=36309,52432,-113561,77732,-117791,-88850,0
C00764=40963,49094,-123815,71578,-117198,-92416,0
C00765=39957,48688,-125104,72501,-116408,-92689,0
C00766=35346,52002,-114801,78562,-117012,-89109,0
C00767=36231,52396,-113664,77798,-117726,-88871,0
C00768=35616,52728,-112686,78546,-117631,-88514,0
C00769=36489,53140,-111514,77810,-118362,-88271,0
C00770=42192,49058,-123959,70243,-117647,-92602,0
C00771=39824,48112,-126997,72427,-115792,-93247,0
C00772=34245,52127,-114412,79731,-116535,-88877,0
C00773=35146,52516,-113293,78948,-117249,-88641,0
C00774=34911,52738,-112646,79266,-117269,-88425,0
C00775=35380,52950,-112040,78867,-117652,-88297,0
C00776=35562,52778,-112540,78619,-117636,-88465,0
C00777=36122,52486,-113400,77942,-117732,-88781,0
C00778=41192,48398,-126080,71061,-116593,-93117,0
C00779=36370,51634,-115908,55379,-126338,-92644,0
C00780=39316,51190,-117293,74145,-118337,-90299,0
C00781=43011,53166,-111573,71101,-121736,-89149,0
C00782=34865,52991,-111914,79402,-117405,-88203,0
C00783=33447,54474,-107676,81337,-117495,-86806,0
C00784=36085,51990,-114849,77799,-117375,-89204,0
C00785=40153,49070,-123874,72437,-116851,-92342,0
C00786=40153,49007,-123894,72446,-116874,-92319,0
C00787=26849,53558,-110019,66755,-124251,-89326,0
C00788=36378,49880,-121062,76771,-116028,-91062,0
C00789=36309,52374,-113580,77741,-117808,-88828,0
C00790=40964,49032,-123834,71587,-117222,-92393,0
C00791=39958,48624,-125124,72509,-116432,-92665,0
C00792=35346,51944,-114819,78571,-117029,-89087,0
C00793=36231,52338,-113682,77807,-117745,-88849,0
C00794=35616,52671,-112705,78555,-117648,-88492,0
C00795=36490,53084,-111533,77819,-118379,-88249,0
C00796=42192,48996,-123979,70253,-117672,-92579,0
C00797=39825,48047,-127016,72435,-115816,-93222,0
C00798=34245,52069,-114431,79740,-116551,-88855,0
C00799=35147,52459,-113311,78957,-117266,-88619,0
C00800=34911,52681,-112664,79274,-117285,-88402,0
C00801=35380,52894,-112059,78875,-117668,-88276,0
C00802=35562,52721,-112558,78628,-117653,-88443,0
C00803=36122,52428,-113418,77951,-117749,-88759,0
C00804=41192,48334,-126099,71070,-116619,-93093,0
C00805=36357,51587,-115891,55414,-126378,-92613,0
C00806=39316,51131,-117312,74155,-118357,-90277,0
C00807=42980,53091,-111645,71137,-121727,-89139,0
C00808=34865,52934,-111932,79411,-117421,-88182,0
C00809=33460,54405,-107734,81329,-117509,-86797,0
C00810=36086,51932,-114868,77808,-117393,-89182,0
C00811=40153,49007,-123894,72446,-116874,-92319,0
C00812=40154,48945,-123913,72454,-116897,-92295,0
C00813=26886,53514,-110002,66734,-124305,-89303,0
C00814=36378,49819,-121081,76780,-116047,-91039,0
C00815=36309,52317,-113598,77750,-117826,-88806,0
C00816=40964,48969,-123854,71596,-117245,-92370,0
C00817=39958,48561,-125142,72518,-116455,-92641,0
C00818=35346,51886,-114838,78580,-117046,-89065,0
C00819=36231,52281,-113701,77816,-117762,-88827,0
C00820=35617,52614,-112723,78564,-117665,-88470,0
C00821=36490,53027,-111551,77828,-118396,-88228,0
C00822=42192,48933,-123998,70262,-117697,-92556,0
C00823=39825,47982,-127036,72444,-115841,-93198,0
C00824=34245,52012,-114449,79748,-116568,-88832,0
C00825=35147,52402,-113330,78966,-117283,-88597,0
C00826=34912,52624,-112683,79283,-117301,-88380,0
C00827=35380,52837,-112077,78884,-117684,-88254,0
C00828=35563,52665,-112577,78637,-117670,-88422,0
C00829=36123,52371,-113437,77960,-117767,-88737,0
C00830=41193,48270,-126119,71079,-116643,-93070,0
C00831=43190,47290,-129457,68527,-116286,-94287,0
C00832=39317,51072,-117330,74164,-118378,-90255,0
C00833=42949,53015,-111717,71172,-121716,-89129,0
C00834=34865,52877,-111951,79420,-117437,-88160,0
C00835=33472,54336,-107791,81321,-117523,-86789,0
C00836=36086,51874,-114886,77817,-117410,-89160,0
C00837=40154,48945,-123913,72454,-116897,-92295,0
C00838=40154,48882,-123932,72464,-116921,-92272,0
C00839=26924,53472,-109984,66713,-124359,-89279,0
C00840=36379,49758,-121100,76788,-116068,-91015,0
C00841=36310,52259,-113616,77759,-117844,-88784,0
C00842=40965,48907,-123873,71605,-117269,-92346,0
C00843=39958,48498,-125161,72527,-116480,-92618,0
C00844=35347,51828,-114856,78589,-117063,-89043,0
C00845=36232,52223,-113719,77825,-117779,-88805,0
C00846=35617,52557,-112741,78573,-117683,-88448,0
C00847=36490,52971,-111569,77838,-118414,-88206,0
C00848=42193,48870,-124018,70271,-117722,-92533,0
C00849=39826,47918,-127055,72452,-115865,-93174,0
C00850=34246,51954,-114468,79756,-116584,-88810,0
C00851=35147,52344,-113348,78975,-117299,-88575,0
C00852=34912,52567,-112701,79292,-117318,-88359,0
C00853=35380,52780,-112095,78893,-117701,-88232,0
C00854=35563,52608,-112595,78646,-117686,-88400,0
C00855=36123,52314,-113455,77969,-117785,-88715,0
C00856=41193,48206,-126138,71088,-116668,-93046,0
C00857=43172,47232,-129447,68560,-116319,-94252,0
C00858=39317,51013,-117348,74174,-118399,-90232,0
C00859=42919,52940,-111789,71207,-121707,-89119,0
C00860=34866,52821,-111969,79429,-117453,-88138,0
C00861=33485,54267,-107848,81312,-117537,-86780,0
C00862=36086,51816,-114905,77826,-117429,-89138,0
C00863=40154,48882,-123932,72464,-116921,-92272,0
C00864=40155,48819,-123951,72473,-116944,-92248,0
C00865=26961,53429,-109966,66692,-124413,-89256,0
C00866=36379,49697,-121119,76797,-116088,-90992,0
C00867=36310,52202,-113635,77768,-117862,-88762,0
C00868=40965,48844,-123892,71614,-117293,-92323,0
C00869=39959,48434,-125181,72536,-116503,-92594,0
C00870=35347,51770,-114875,78598,-117081,-89020,0
C00871=36232,52166,-113738,77834,-117798,-88783,0
C00872=35617,52500,-112760,78582,-117699,-88427,0
C00873=36491,52914,-111588,77847,-118431,-88184,0
C00874=42193,48808,-124036,70281,-117747,-92510,0
C00875=39826,47853,-127074,72461,-115889,-93150,0
C00876=34246,51896,-114486,79765,-116600,-88788,0
C00877=35148,52287,-113366,78984,-117316,-88553,0
C00878=34912,52510,-112719,79301,-117335,-88337,0
C00879=35381,52723,-112114,78902,-117718,-88210,0
C00880=35563,52551,-112613,78655,-117703,-88378,0
C00881=36123,52256,-113473,77978,-117802,-88693,0
C00882=41193,48142,-126158,71097,-116693,-93022,0
C00883=43153,47175,-129436,68593,-116350,-94217,0
C00884=39317,50954,-117367,74183,-118419,-90210,0
C00885=42888,52864,-111861,71243,-121697,-89108,0
C00886=34866,52764,-111987,79437,-117469,-88116,0
C00887=33497,54198,-107905,81304,-117551,-86771,0
C00888=36087,51758,-114924,77835,-117446,-89116,0
C00889=40155,48819,-123951,72473,-116944,-92248,0
C00890=40155,48757,-123970,72482,-116967,-92225,0
C00891=26998,53386,-109948,66671,-124467,-89232,0
C00892=36379,49636,-121137,76805,-116107,-90969,0
C00893=36310,52145,-113653,77777,-117879,-88740,0
C00894=40965,48782,-123911,71624,-117317,-92300,0
C00895=39959,48371,-125199,72545,-116527,-92570,0
C00896=35347,51712,-114893,78606,-117098,-88998,0
C00897=36232,52109,-113756,77844,-117815,-88761,0
C00898=35618,52443,-112778,78591,-117716,-88405,0
C00899=36491,52858,-111606,77856,-118448,-88163,0
C00900=42194,48745,-124056,70290,-117771,-92486,0
C00901=39826,47789,-127093,72469,-115913,-93125,0
C00902=34246,51838,-114505,79773,-116617,-88766,0
C00903=35148,52230,-113385,78992,-117333,-88531,0
C00904=34913,52453,-112738,79310,-117352,-88315,0
C00905=35381,52667,-112132,78911,-117734,-88189,0
C00906=35564,52494,-112631,78664,-117721,-88355,0
C00907=36124,52199,-113492,77987,-117819,-88671,0
C00908=41194,48078,-126177,71106,-116717,-92998,0
C00909=43135,47117,-129426,68626,-116381,-94181,0
C00910=39318,50894,-117385,74193,-118440,-90187,0
C00911=42857,52789,-111933,71278,-121688,-89098,0
C00912=34866,52707,-112006,79446,-117485,-88094,0
C00913=33510,54129,-107962,81296,-117566,-86763,0
C00914=36087,51700,-114942,77844,-117464,-89094,0
C00915=40155,48757,-123970,72482,-116967,-92225,0
C00916=40156,48694,-123989,72491,-116991,-92201,0
C00917=27036,53343,-109930,66650,-124521,-89208,0
C00918=36380,49575,-121157,76814,-116127,-90945,0
C00919=36311,52087,-113671,77786,-117896,-88718,0
C00920=40966,48719,-123930,71633,-117341,-92276,0
C00921=39960,48308,-125219,72554,-116551,-92546,0
C00922=35348,51654,-114911,78615,-117115,-88975,0
C00923=36233,52051,-113774,77853,-117832,-88739,0
C00924=35618,52386,-112796,78600,-117733,-88383,0
C00925=36491,52801,-111624,77866,-118465,-88141,0
C00926=42194,48682,-124074,70300,-117796,-92463,0
C00927=39827,47725,-127113,72478,-115937,-93101,0
C00928=34247,51781,-114523,79782,-116634,-88743,0
C00929=35148,52173,-113403,79001,-117349,-88509,0
C00930=34913,52396,-112756,79318,-117368,-88293,0
C00931=35381,52610,-112150,78920,-117752,-88167,0
C00932=35564,52437,-112650,78673,-117738,-88334,0
C00933=36124,52142,-113510,77997,-117837,-88649,0
C00934=41194,48015,-126196,71115,-116743,-92974,0
C00935=43116,47060,-129416,68659,-116412,-94147,0
C00936=39318,50835,-117403,74203,-118461,-90165,0
C00937=42826,52713,-112005,71313,-121678,-89087,0
C00938=34867,52651,-112024,79455,-117502,-88072,0
C00939=33523,54060,-108019,81288,-117579,-86755,0
C00940=36088,51643,-114959,77853,-117483,-89071,0
C00941=40156,48694,-123989,72491,-116991,-92201,0
C00942=40156,48632,-124008,72500,-117014,-92178,0
C00943=27073,53300,-109912,66630,-124575,-89185,0
//INST
///DATE 2025/02/20 16:20
///COMM Generated using RoboDK
///ATTR SC,RW
///GROUP1 RB1
NOP
MOVL C00000 V=130.0 PL=1
MOVL C00001 V=30.0 PL=1
MOVL C00002 V=130.0 PL=1
MOVL C00003 V=30.0 PL=1
MOVL C00004 V=130.0 PL=1
MOVL C00005 V=20.0 PL=1
MOVL C00006 V=130.0 PL=1
MOVL C00007 V=130.0 PL=1
MOVL C00008 V=30.0 PL=1
MOVL C00009 V=130.0 PL=1
MOVL C00010 V=60.0 PL=1
MOVL C00011 V=60.0 PL=1
MOVL C00012 V=60.0 PL=1
MOVL C00013 V=60.0 PL=1
MOVL C00014 V=130.0 PL=1
MOVL C00015 V=30.0 PL=1
MOVL C00016 V=30.0 PL=1
MOVL C00017 V=30.0 PL=1
MOVL C00018 V=30.0 PL=1
MOVL C00019 V=30.0 PL=1
MOVL C00020 V=30.0 PL=1
MOVL C00021 V=30.0 PL=1
MOVL C00022 V=30.0 PL=1
MOVL C00023 V=130.0 PL=1
MOVL C00024 V=130.0 PL=1
MOVL C00025 V=30.0 PL=1
MOVL C00026 V=130.0 PL=1
MOVL C00027 V=30.0 PL=1
MOVL C00028 V=130.0 PL=1
MOVL C00029 V=30.0 PL=1
MOVL C00030 V=130.0 PL=1
MOVL C00031 V=20.0 PL=1
MOVL C00032 V=130.0 PL=1
MOVL C00033 V=130.0 PL=1
MOVL C00034 V=30.0 PL=1
MOVL C00035 V=130.0 PL=1
MOVL C00036 V=60.0 PL=1
MOVL C00037 V=60.0 PL=1
MOVL C00038 V=60.0 PL=1
MOVL C00039 V=60.0 PL=1
MOVL C00040 V=130.0 PL=1
MOVL C00041 V=30.0 PL=1
MOVL C00042 V=30.0 PL=1
MOVL C00043 V=30.0 PL=1
MOVL C00044 V=30.0 PL=1
MOVL C00045 V=30.0 PL=1
MOVL C00046 V=30.0 PL=1
MOVL C00047 V=30.0 PL=1
MOVL C00048 V=30.0 PL=1
MOVL C00049 V=130.0 PL=1
MOVL C00050 V=130.0 PL=1
MOVL C00051 V=30.0 PL=1
MOVL C00052 V=130.0 PL=1
MOVL C00053 V=30.0 PL=1
MOVL C00054 V=130.0 PL=1
MOVL C00055 V=30.0 PL=1
MOVL C00056 V=130.0 PL=1
MOVL C00057 V=20.0 PL=1
MOVL C00058 V=130.0 PL=1
MOVL C00059 V=130.0 PL=1
MOVL C00060 V=30.0 PL=1
MOVL C00061 V=130.0 PL=1
MOVL C00062 V=60.0 PL=1
MOVL C00063 V=60.0 PL=1
MOVL C00064 V=60.0 PL=1
MOVL C00065 V=60.0 PL=1
MOVL C00066 V=130.0 PL=1
MOVL C00067 V=30.0 PL=1
MOVL C00068 V=30.0 PL=1
MOVL C00069 V=30.0 PL=1
MOVL C00070 V=30.0 PL=1
MOVL C00071 V=30.0 PL=1
MOVL C00072 V=30.0 PL=1
MOVL C00073 V=30.0 PL=1
MOVL C00074 V=30.0 PL=1
MOVL C00075 V=130.0 PL=1
MOVL C00076 V=130.0 PL=1
MOVL C00077 V=30.0 PL=1
MOVL C00078 V=130.0 PL=1
MOVL C00079 V=30.0 PL=1
MOVL C00080 V=130.0 PL=1
MOVL C00081 V=30.0 PL=1
MOVL C00082 V=130.0 PL=1
MOVL C00083 V=20.0 PL=1
MOVL C00084 V=130.0 PL=1
MOVL C00085 V=130.0 PL=1
MOVL C00086 V=30.0 PL=1
MOVL C00087 V=130.0 PL=1
MOVL C00088 V=60.0 PL=1
MOVL C00089 V=60.0 PL=1
MOVL C00090 V=60.0 PL=1
MOVL C00091 V=60.0 PL=1
MOVL C00092 V=130.0 PL=1
MOVL C00093 V=30.0 PL=1
MOVL C00094 V=30.0 PL=1
MOVL C00095 V=30.0 PL=1
MOVL C00096 V=30.0 PL=1
MOVL C00097 V=30.0 PL=1
MOVL C00098 V=30.0 PL=1
MOVL C00099 V=30.0 PL=1
MOVL C00100 V=30.0 PL=1
MOVL C00101 V=130.0 PL=1
MOVL C00102 V=130.0 PL=1
MOVL C00103 V=30.0 PL=1
MOVL C00104 V=130.0 PL=1
MOVL C00105 V=30.0 PL=1
MOVL C00106 V=130.0 PL=1
MOVL C00107 V=30.0 PL=1
MOVL C00108 V=130.0 PL=1
MOVL C00109 V=20.0 PL=1
MOVL C00110 V=130.0 PL=1
MOVL C00111 V=130.0 PL=1
MOVL C00112 V=30.0 PL=1
MOVL C00113 V=130.0 PL=1
MOVL C00114 V=60.0 PL=1
MOVL C00115 V=60.0 PL=1
MOVL C00116 V=60.0 PL=1
MOVL C00117 V=60.0 PL=1
MOVL C00118 V=130.0 PL=1
MOVL C00119 V=30.0 PL=1
MOVL C00120 V=30.0 PL=1
MOVL C00121 V=30.0 PL=1
MOVL C00122 V=30.0 PL=1
MOVL C00123 V=30.0 PL=1
MOVL C00124 V=30.0 PL=1
MOVL C00125 V=30.0 PL=1
MOVL C00126 V=30.0 PL=1
MOVL C00127 V=130.0 PL=1
MOVL C00128 V=130.0 PL=1
MOVL C00129 V=30.0 PL=1
MOVL C00130 V=130.0 PL=1
MOVL C00131 V=30.0 PL=1
MOVL C00132 V=130.0 PL=1
MOVL C00133 V=30.0 PL=1
MOVL C00134 V=130.0 PL=1
MOVL C00135 V=20.0 PL=1
MOVL C00136 V=130.0 PL=1
MOVL C00137 V=130.0 PL=1
MOVL C00138 V=30.0 PL=1
MOVL C00139 V=130.0 PL=1
MOVL C00140 V=60.0 PL=1
MOVL C00141 V=60.0 PL=1
MOVL C00142 V=60.0 PL=1
MOVL C00143 V=60.0 PL=1
MOVL C00144 V=130.0 PL=1
MOVL C00145 V=30.0 PL=1
MOVL C00146 V=30.0 PL=1
MOVL C00147 V=30.0 PL=1
MOVL C00148 V=30.0 PL=1
MOVL C00149 V=30.0 PL=1
MOVL C00150 V=30.0 PL=1
MOVL C00151 V=30.0 PL=1
MOVL C00152 V=30.0 PL=1
MOVL C00153 V=130.0 PL=1
MOVL C00154 V=130.0 PL=1
MOVL C00155 V=30.0 PL=1
MOVL C00156 V=130.0 PL=1
MOVL C00157 V=30.0 PL=1
MOVL C00158 V=130.0 PL=1
MOVL C00159 V=30.0 PL=1
MOVL C00160 V=130.0 PL=1
MOVL C00161 V=20.0 PL=1
MOVL C00162 V=130.0 PL=1
MOVL C00163 V=130.0 PL=1
MOVL C00164 V=30.0 PL=1
MOVL C00165 V=130.0 PL=1
MOVL C00166 V=60.0 PL=1
MOVL C00167 V=60.0 PL=1
MOVL C00168 V=60.0 PL=1
MOVL C00169 V=60.0 PL=1
MOVL C00170 V=130.0 PL=1
MOVL C00171 V=30.0 PL=1
MOVL C00172 V=30.0 PL=1
MOVL C00173 V=30.0 PL=1
MOVL C00174 V=30.0 PL=1
MOVL C00175 V=30.0 PL=1
MOVL C00176 V=30.0 PL=1
MOVL C00177 V=30.0 PL=1
MOVL C00178 V=30.0 PL=1
MOVL C00179 V=130.0 PL=1
MOVL C00180 V=130.0 PL=1
MOVL C00181 V=30.0 PL=1
MOVL C00182 V=130.0 PL=1
MOVL C00183 V=30.0 PL=1
MOVL C00184 V=130.0 PL=1
MOVL C00185 V=30.0 PL=1
MOVL C00186 V=130.0 PL=1
MOVL C00187 V=20.0 PL=1
MOVL C00188 V=130.0 PL=1
MOVL C00189 V=130.0 PL=1
MOVL C00190 V=30.0 PL=1
MOVL C00191 V=130.0 PL=1
MOVL C00192 V=60.0 PL=1
MOVL C00193 V=60.0 PL=1
MOVL C00194 V=60.0 PL=1
MOVL C00195 V=60.0 PL=1
MOVL C00196 V=130.0 PL=1
MOVL C00197 V=30.0 PL=1
MOVL C00198 V=30.0 PL=1
MOVL C00199 V=30.0 PL=1
MOVL C00200 V=30.0 PL=1
MOVL C00201 V=30.0 PL=1
MOVL C00202 V=30.0 PL=1
MOVL C00203 V=30.0 PL=1
MOVL C00204 V=30.0 PL=1
MOVL C00205 V=130.0 PL=1
MOVL C00206 V=130.0 PL=1
MOVL C00207 V=30.0 PL=1
MOVL C00208 V=130.0 PL=1
MOVL C00209 V=30.0 PL=1
MOVL C00210 V=130.0 PL=1
MOVL C00211 V=30.0 PL=1
MOVL C00212 V=130.0 PL=1
MOVL C00213 V=20.0 PL=1
MOVL C00214 V=130.0 PL=1
MOVL C00215 V=130.0 PL=1
MOVL C00216 V=30.0 PL=1
MOVL C00217 V=130.0 PL=1
MOVL C00218 V=60.0 PL=1
MOVL C00219 V=60.0 PL=1
MOVL C00220 V=60.0 PL=1
MOVL C00221 V=60.0 PL=1
MOVL C00222 V=130.0 PL=1
MOVL C00223 V=30.0 PL=1
MOVL C00224 V=30.0 PL=1
MOVL C00225 V=30.0 PL=1
MOVL C00226 V=30.0 PL=1
MOVL C00227 V=30.0 PL=1
MOVL C00228 V=30.0 PL=1
MOVL C00229 V=30.0 PL=1
MOVL C00230 V=30.0 PL=1
MOVL C00231 V=130.0 PL=1
MOVL C00232 V=130.0 PL=1
MOVL C00233 V=30.0 PL=1
MOVL C00234 V=130.0 PL=1
MOVL C00235 V=30.0 PL=1
MOVL C00236 V=130.0 PL=1
MOVL C00237 V=30.0 PL=1
MOVL C00238 V=130.0 PL=1
MOVL C00239 V=20.0 PL=1
MOVL C00240 V=130.0 PL=1
MOVL C00241 V=130.0 PL=1
MOVL C00242 V=30.0 PL=1
MOVL C00243 V=130.0 PL=1
MOVL C00244 V=60.0 PL=1
MOVL C00245 V=60.0 PL=1
MOVL C00246 V=60.0 PL=1
MOVL C00247 V=60.0 PL=1
MOVL C00248 V=130.0 PL=1
MOVL C00249 V=30.0 PL=1
MOVL C00250 V=30.0 PL=1
MOVL C00251 V=30.0 PL=1
MOVL C00252 V=30.0 PL=1
MOVL C00253 V=30.0 PL=1
MOVL C00254 V=30.0 PL=1
MOVL C00255 V=30.0 PL=1
MOVL C00256 V=30.0 PL=1
MOVL C00257 V=130.0 PL=1
MOVL C00258 V=130.0 PL=1
MOVL C00259 V=30.0 PL=1
MOVL C00260 V=130.0 PL=1
MOVL C00261 V=30.0 PL=1
MOVL C00262 V=130.0 PL=1
MOVL C00263 V=30.0 PL=1
MOVL C00264 V=130.0 PL=1
MOVL C00265 V=20.0 PL=1
MOVL C00266 V=130.0 PL=1
MOVL C00267 V=130.0 PL=1
MOVL C00268 V=30.0 PL=1
MOVL C00269 V=130.0 PL=1
MOVL C00270 V=60.0 PL=1
MOVL C00271 V=60.0 PL=1
MOVL C00272 V=60.0 PL=1
MOVL C00273 V=60.0 PL=1
MOVL C00274 V=130.0 PL=1
MOVL C00275 V=30.0 PL=1
MOVL C00276 V=30.0 PL=1
MOVL C00277 V=30.0 PL=1
MOVL C00278 V=30.0 PL=1
MOVL C00279 V=30.0 PL=1
MOVL C00280 V=30.0 PL=1
MOVL C00281 V=30.0 PL=1
MOVL C00282 V=30.0 PL=1
MOVL C00283 V=130.0 PL=1
MOVL C00284 V=130.0 PL=1
MOVL C00285 V=30.0 PL=1
MOVL C00286 V=130.0 PL=1
MOVL C00287 V=30.0 PL=1
MOVL C00288 V=130.0 PL=1
MOVL C00289 V=30.0 PL=1
MOVL C00290 V=130.0 PL=1
MOVL C00291 V=20.0 PL=1
MOVL C00292 V=130.0 PL=1
MOVL C00293 V=130.0 PL=1
MOVL C00294 V=30.0 PL=1
MOVL C00295 V=130.0 PL=1
MOVL C00296 V=60.0 PL=1
MOVL C00297 V=60.0 PL=1
MOVL C00298 V=60.0 PL=1
MOVL C00299 V=60.0 PL=1
MOVL C00300 V=130.0 PL=1
MOVL C00301 V=30.0 PL=1
MOVL C00302 V=30.0 PL=1
MOVL C00303 V=30.0 PL=1
MOVL C00304 V=30.0 PL=1
MOVL C00305 V=30.0 PL=1
MOVL C00306 V=30.0 PL=1
MOVL C00307 V=30.0 PL=1
MOVL C00308 V=30.0 PL=1
MOVL C00309 V=130.0 PL=1
MOVL C00310 V=130.0 PL=1
MOVL C00311 V=30.0 PL=1
MOVL C00312 V=130.0 PL=1
MOVL C00313 V=30.0 PL=1
MOVL C00314 V=130.0 PL=1
MOVL C00315 V=30.0 PL=1
MOVL C00316 V=130.0 PL=1
MOVL C00317 V=20.0 PL=1
MOVL C00318 V=130.0 PL=1
MOVL C00319 V=130.0 PL=1
MOVL C00320 V=30.0 PL=1
MOVL C00321 V=130.0 PL=1
MOVL C00322 V=60.0 PL=1
MOVL C00323 V=60.0 PL=1
MOVL C00324 V=60.0 PL=1
MOVL C00325 V=60.0 PL=1
MOVL C00326 V=130.0 PL=1
MOVL C00327 V=30.0 PL=1
MOVL C00328 V=30.0 PL=1
MOVL C00329 V=30.0 PL=1
MOVL C00330 V=30.0 PL=1
MOVL C00331 V=30.0 PL=1
MOVL C00332 V=30.0 PL=1
MOVL C00333 V=30.0 PL=1
MOVL C00334 V=30.0 PL=1
MOVL C00335 V=130.0 PL=1
MOVL C00336 V=130.0 PL=1
MOVL C00337 V=30.0 PL=1
MOVL C00338 V=130.0 PL=1
MOVL C00339 V=30.0 PL=1
MOVL C00340 V=130.0 PL=1
MOVL C00341 V=30.0 PL=1
MOVL C00342 V=130.0 PL=1
MOVL C00343 V=20.0 PL=1
MOVL C00344 V=130.0 PL=1
MOVL C00345 V=130.0 PL=1
MOVL C00346 V=30.0 PL=1
MOVL C00347 V=130.0 PL=1
MOVL C00348 V=60.0 PL=1
MOVL C00349 V=60.0 PL=1
MOVL C00350 V=60.0 PL=1
MOVL C00351 V=60.0 PL=1
MOVL C00352 V=130.0 PL=1
MOVL C00353 V=30.0 PL=1
MOVL C00354 V=30.0 PL=1
MOVL C00355 V=30.0 PL=1
MOVL C00356 V=30.0 PL=1
MOVL C00357 V=30.0 PL=1
MOVL C00358 V=30.0 PL=1
MOVL C00359 V=30.0 PL=1
MOVL C00360 V=30.0 PL=1
MOVL C00361 V=130.0 PL=1
MOVL C00362 V=130.0 PL=1
MOVL C00363 V=30.0 PL=1
MOVL C00364 V=130.0 PL=1
MOVL C00365 V=30.0 PL=1
MOVL C00366 V=130.0 PL=1
MOVL C00367 V=30.0 PL=1
MOVL C00368 V=130.0 PL=1
MOVL C00369 V=20.0 PL=1
MOVL C00370 V=130.0 PL=1
MOVL C00371 V=130.0 PL=1
MOVL C00372 V=30.0 PL=1
MOVL C00373 V=130.0 PL=1
MOVL C00374 V=60.0 PL=1
MOVL C00375 V=60.0 PL=1
MOVL C00376 V=60.0 PL=1
MOVL C00377 V=60.0 PL=1
MOVL C00378 V=130.0 PL=1
MOVL C00379 V=30.0 PL=1
MOVL C00380 V=30.0 PL=1
MOVL C00381 V=30.0 PL=1
MOVL C00382 V=30.0 PL=1
MOVL C00383 V=30.0 PL=1
MOVL C00384 V=30.0 PL=1
MOVL C00385 V=30.0 PL=1
MOVL C00386 V=30.0 PL=1
MOVL C00387 V=130.0 PL=1
MOVL C00388 V=130.0 PL=1
MOVL C00389 V=30.0 PL=1
MOVL C00390 V=130.0 PL=1
MOVL C00391 V=30.0 PL=1
MOVL C00392 V=130.0 PL=1
MOVL C00393 V=30.0 PL=1
MOVL C00394 V=130.0 PL=1
MOVL C00395 V=20.0 PL=1
MOVL C00396 V=130.0 PL=1
MOVL C00397 V=130.0 PL=1
MOVL C00398 V=30.0 PL=1
MOVL C00399 V=130.0 PL=1
MOVL C00400 V=60.0 PL=1
MOVL C00401 V=60.0 PL=1
MOVL C00402 V=60.0 PL=1
MOVL C00403 V=60.0 PL=1
MOVL C00404 V=130.0 PL=1
MOVL C00405 V=30.0 PL=1
MOVL C00406 V=30.0 PL=1
MOVL C00407 V=30.0 PL=1
MOVL C00408 V=30.0 PL=1
MOVL C00409 V=30.0 PL=1
MOVL C00410 V=30.0 PL=1
MOVL C00411 V=30.0 PL=1
MOVL C00412 V=30.0 PL=1
MOVL C00413 V=130.0 PL=1
MOVL C00414 V=130.0 PL=1
MOVL C00415 V=30.0 PL=1
MOVL C00416 V=130.0 PL=1
MOVL C00417 V=30.0 PL=1
MOVL C00418 V=130.0 PL=1
MOVL C00419 V=30.0 PL=1
MOVL C00420 V=130.0 PL=1
MOVL C00421 V=20.0 PL=1
MOVL C00422 V=130.0 PL=1
MOVL C00423 V=130.0 PL=1
MOVL C00424 V=30.0 PL=1
MOVL C00425 V=130.0 PL=1
MOVL C00426 V=60.0 PL=1
MOVL C00427 V=60.0 PL=1
MOVL C00428 V=60.0 PL=1
MOVL C00429 V=60.0 PL=1
MOVL C00430 V=130.0 PL=1
MOVL C00431 V=30.0 PL=1
MOVL C00432 V=30.0 PL=1
MOVL C00433 V=30.0 PL=1
MOVL C00434 V=30.0 PL=1
MOVL C00435 V=30.0 PL=1
MOVL C00436 V=30.0 PL=1
MOVL C00437 V=30.0 PL=1
MOVL C00438 V=30.0 PL=1
MOVL C00439 V=130.0 PL=1
MOVL C00440 V=130.0 PL=1
MOVL C00441 V=30.0 PL=1
MOVL C00442 V=130.0 PL=1
MOVL C00443 V=30.0 PL=1
MOVL C00444 V=130.0 PL=1
MOVL C00445 V=30.0 PL=1
MOVL C00446 V=130.0 PL=1
MOVL C00447 V=20.0 PL=1
MOVL C00448 V=130.0 PL=1
MOVL C00449 V=130.0 PL=1
MOVL C00450 V=30.0 PL=1
MOVL C00451 V=130.0 PL=1
MOVL C00452 V=60.0 PL=1
MOVL C00453 V=60.0 PL=1
MOVL C00454 V=60.0 PL=1
MOVL C00455 V=60.0 PL=1
MOVL C00456 V=130.0 PL=1
MOVL C00457 V=30.0 PL=1
MOVL C00458 V=30.0 PL=1
MOVL C00459 V=30.0 PL=1
MOVL C00460 V=30.0 PL=1
MOVL C00461 V=30.0 PL=1
MOVL C00462 V=30.0 PL=1
MOVL C00463 V=30.0 PL=1
MOVL C00464 V=30.0 PL=1
MOVL C00465 V=130.0 PL=1
MOVL C00466 V=130.0 PL=1
MOVL C00467 V=30.0 PL=1
MOVL C00468 V=130.0 PL=1
MOVL C00469 V=30.0 PL=1
MOVL C00470 V=130.0 PL=1
MOVL C00471 V=30.0 PL=1
MOVL C00472 V=130.0 PL=1
MOVL C00473 V=20.0 PL=1
MOVL C00474 V=130.0 PL=1
MOVL C00475 V=130.0 PL=1
MOVL C00476 V=30.0 PL=1
MOVL C00477 V=130.0 PL=1
MOVL C00478 V=60.0 PL=1
MOVL C00479 V=60.0 PL=1
MOVL C00480 V=60.0 PL=1
MOVL C00481 V=60.0 PL=1
MOVL C00482 V=130.0 PL=1
MOVL C00483 V=30.0 PL=1
MOVL C00484 V=30.0 PL=1
MOVL C00485 V=30.0 PL=1
MOVL C00486 V=30.0 PL=1
MOVL C00487 V=30.0 PL=1
MOVL C00488 V=30.0 PL=1
MOVL C00489 V=30.0 PL=1
MOVL C00490 V=30.0 PL=1
MOVL C00491 V=130.0 PL=1
MOVL C00492 V=130.0 PL=1
MOVL C00493 V=30.0 PL=1
MOVL C00494 V=130.0 PL=1
MOVL C00495 V=30.0 PL=1
MOVL C00496 V=130.0 PL=1
MOVL C00497 V=30.0 PL=1
MOVL C00498 V=130.0 PL=1
MOVL C00499 V=20.0 PL=1
MOVL C00500 V=130.0 PL=1
MOVL C00501 V=130.0 PL=1
MOVL C00502 V=30.0 PL=1
MOVL C00503 V=130.0 PL=1
MOVL C00504 V=60.0 PL=1
MOVL C00505 V=60.0 PL=1
MOVL C00506 V=60.0 PL=1
MOVL C00507 V=60.0 PL=1
MOVL C00508 V=130.0 PL=1
MOVL C00509 V=30.0 PL=1
MOVL C00510 V=30.0 PL=1
MOVL C00511 V=30.0 PL=1
MOVL C00512 V=30.0 PL=1
MOVL C00513 V=30.0 PL=1
MOVL C00514 V=30.0 PL=1
MOVL C00515 V=30.0 PL=1
MOVL C00516 V=30.0 PL=1
MOVL C00517 V=130.0 PL=1
MOVL C00518 V=130.0 PL=1
MOVL C00519 V=30.0 PL=1
MOVL C00520 V=130.0 PL=1
MOVL C00521 V=30.0 PL=1
MOVL C00522 V=130.0 PL=1
MOVL C00523 V=30.0 PL=1
MOVL C00524 V=130.0 PL=1
MOVL C00525 V=20.0 PL=1
MOVL C00526 V=130.0 PL=1
MOVL C00527 V=130.0 PL=1
MOVL C00528 V=30.0 PL=1
MOVL C00529 V=130.0 PL=1
MOVL C00530 V=60.0 PL=1
MOVL C00531 V=60.0 PL=1
MOVL C00532 V=60.0 PL=1
MOVL C00533 V=60.0 PL=1
MOVL C00534 V=130.0 PL=1
MOVL C00535 V=30.0 PL=1
MOVL C00536 V=30.0 PL=1
MOVL C00537 V=30.0 PL=1
MOVL C00538 V=30.0 PL=1
MOVL C00539 V=30.0 PL=1
MOVL C00540 V=30.0 PL=1
MOVL C00541 V=30.0 PL=1
MOVL C00542 V=30.0 PL=1
MOVL C00543 V=130.0 PL=1
MOVL C00544 V=130.0 PL=1
MOVL C00545 V=30.0 PL=1
MOVL C00546 V=130.0 PL=1
MOVL C00547 V=30.0 PL=1
MOVL C00548 V=130.0 PL=1
MOVL C00549 V=30.0 PL=1
MOVL C00550 V=130.0 PL=1
MOVL C00551 V=20.0 PL=1
MOVL C00552 V=130.0 PL=1
MOVL C00553 V=130.0 PL=1
MOVL C00554 V=30.0 PL=1
MOVL C00555 V=130.0 PL=1
MOVL C00556 V=60.0 PL=1
MOVL C00557 V=60.0 PL=1
MOVL C00558 V=60.0 PL=1
MOVL C00559 V=60.0 PL=1
MOVL C00560 V=130.0 PL=1
MOVL C00561 V=30.0 PL=1
MOVL C00562 V=30.0 PL=1
MOVL C00563 V=30.0 PL=1
MOVL C00564 V=30.0 PL=1
MOVL C00565 V=30.0 PL=1
MOVL C00566 V=30.0 PL=1
MOVL C00567 V=30.0 PL=1
MOVL C00568 V=30.0 PL=1
MOVL C00569 V=130.0 PL=1
MOVL C00570 V=130.0 PL=1
MOVL C00571 V=30.0 PL=1
MOVL C00572 V=130.0 PL=1
MOVL C00573 V=30.0 PL=1
MOVL C00574 V=130.0 PL=1
MOVL C00575 V=30.0 PL=1
MOVL C00576 V=130.0 PL=1
MOVL C00577 V=20.0 PL=1
MOVL C00578 V=130.0 PL=1
MOVL C00579 V=130.0 PL=1
MOVL C00580 V=30.0 PL=1
MOVL C00581 V=130.0 PL=1
MOVL C00582 V=60.0 PL=1
MOVL C00583 V=60.0 PL=1
MOVL C00584 V=60.0 PL=1
MOVL C00585 V=60.0 PL=1
MOVL C00586 V=130.0 PL=1
MOVL C00587 V=30.0 PL=1
MOVL C00588 V=30.0 PL=1
MOVL C00589 V=30.0 PL=1
MOVL C00590 V=30.0 PL=1
MOVL C00591 V=30.0 PL=1
MOVL C00592 V=30.0 PL=1
MOVL C00593 V=30.0 PL=1
MOVL C00594 V=30.0 PL=1
MOVL C00595 V=130.0 PL=1
MOVL C00596 V=130.0 PL=1
MOVL C00597 V=30.0 PL=1
MOVL C00598 V=130.0 PL=1
MOVL C00599 V=30.0 PL=1
MOVL C00600 V=130.0 PL=1
MOVL C00601 V=30.0 PL=1
MOVL C00602 V=130.0 PL=1
MOVL C00603 V=20.0 PL=1
MOVL C00604 V=130.0 PL=1
MOVL C00605 V=130.0 PL=1
MOVL C00606 V=30.0 PL=1
MOVL C00607 V=130.0 PL=1
MOVL C00608 V=60.0 PL=1
MOVL C00609 V=60.0 PL=1
MOVL C00610 V=60.0 PL=1
MOVL C00611 V=60.0 PL=1
MOVL C00612 V=130.0 PL=1
MOVL C00613 V=30.0 PL=1
MOVL C00614 V=30.0 PL=1
MOVL C00615 V=30.0 PL=1
MOVL C00616 V=30.0 PL=1
MOVL C00617 V=30.0 PL=1
MOVL C00618 V=30.0 PL=1
MOVL C00619 V=30.0 PL=1
MOVL C00620 V=30.0 PL=1
MOVL C00621 V=130.0 PL=1
MOVL C00622 V=130.0 PL=1
MOVL C00623 V=30.0 PL=1
MOVL C00624 V=130.0 PL=1
MOVL C00625 V=30.0 PL=1
MOVL C00626 V=130.0 PL=1
MOVL C00627 V=30.0 PL=1
MOVL C00628 V=130.0 PL=1
MOVL C00629 V=20.0 PL=1
MOVL C00630 V=130.0 PL=1
MOVL C00631 V=130.0 PL=1
MOVL C00632 V=30.0 PL=1
MOVL C00633 V=130.0 PL=1
MOVL C00634 V=60.0 PL=1
MOVL C00635 V=60.0 PL=1
MOVL C00636 V=60.0 PL=1
MOVL C00637 V=60.0 PL=1
MOVL C00638 V=130.0 PL=1
MOVL C00639 V=30.0 PL=1
MOVL C00640 V=30.0 PL=1
MOVL C00641 V=30.0 PL=1
MOVL C00642 V=30.0 PL=1
MOVL C00643 V=30.0 PL=1
MOVL C00644 V=30.0 PL=1
MOVL C00645 V=30.0 PL=1
MOVL C00646 V=30.0 PL=1
MOVL C00647 V=130.0 PL=1
MOVL C00648 V=130.0 PL=1
MOVL C00649 V=30.0 PL=1
MOVL C00650 V=130.0 PL=1
MOVL C00651 V=30.0 PL=1
MOVL C00652 V=130.0 PL=1
MOVL C00653 V=30.0 PL=1
MOVL C00654 V=130.0 PL=1
MOVL C00655 V=20.0 PL=1
MOVL C00656 V=130.0 PL=1
MOVL C00657 V=130.0 PL=1
MOVL C00658 V=30.0 PL=1
MOVL C00659 V=130.0 PL=1
MOVL C00660 V=60.0 PL=1
MOVL C00661 V=60.0 PL=1
MOVL C00662 V=60.0 PL=1
MOVL C00663 V=60.0 PL=1
MOVL C00664 V=130.0 PL=1
MOVL C00665 V=30.0 PL=1
MOVL C00666 V=30.0 PL=1
MOVL C00667 V=30.0 PL=1
MOVL C00668 V=30.0 PL=1
MOVL C00669 V=30.0 PL=1
MOVL C00670 V=30.0 PL=1
MOVL C00671 V=30.0 PL=1
MOVL C00672 V=30.0 PL=1
MOVL C00673 V=130.0 PL=1
MOVL C00674 V=130.0 PL=1
MOVL C00675 V=30.0 PL=1
MOVL C00676 V=130.0 PL=1
MOVL C00677 V=30.0 PL=1
MOVL C00678 V=130.0 PL=1
MOVL C00679 V=30.0 PL=1
MOVL C00680 V=130.0 PL=1
MOVL C00681 V=20.0 PL=1
MOVL C00682 V=130.0 PL=1
MOVL C00683 V=130.0 PL=1
MOVL C00684 V=30.0 PL=1
MOVL C00685 V=130.0 PL=1
MOVL C00686 V=60.0 PL=1
MOVL C00687 V=60.0 PL=1
MOVL C00688 V=60.0 PL=1
MOVL C00689 V=60.0 PL=1
MOVL C00690 V=130.0 PL=1
MOVL C00691 V=30.0 PL=1
MOVL C00692 V=30.0 PL=1
MOVL C00693 V=30.0 PL=1
MOVL C00694 V=30.0 PL=1
MOVL C00695 V=30.0 PL=1
MOVL C00696 V=30.0 PL=1
MOVL C00697 V=30.0 PL=1
MOVL C00698 V=30.0 PL=1
MOVL C00699 V=130.0 PL=1
MOVL C00700 V=130.0 PL=1
MOVL C00701 V=30.0 PL=1
MOVL C00702 V=130.0 PL=1
MOVL C00703 V=30.0 PL=1
MOVL C00704 V=130.0 PL=1
MOVL C00705 V=30.0 PL=1
MOVL C00706 V=130.0 PL=1
MOVL C00707 V=20.0 PL=1
MOVL C00708 V=130.0 PL=1
MOVL C00709 V=130.0 PL=1
MOVL C00710 V=30.0 PL=1
MOVL C00711 V=130.0 PL=1
MOVL C00712 V=60.0 PL=1
MOVL C00713 V=60.0 PL=1
MOVL C00714 V=60.0 PL=1
MOVL C00715 V=60.0 PL=1
MOVL C00716 V=130.0 PL=1
MOVL C00717 V=30.0 PL=1
MOVL C00718 V=30.0 PL=1
MOVL C00719 V=30.0 PL=1
MOVL C00720 V=30.0 PL=1
MOVL C00721 V=30.0 PL=1
MOVL C00722 V=30.0 PL=1
MOVL C00723 V=30.0 PL=1
MOVL C00724 V=30.0 PL=1
MOVL C00725 V=130.0 PL=1
MOVL C00726 V=130.0 PL=1
MOVL C00727 V=30.0 PL=1
MOVL C00728 V=130.0 PL=1
MOVL C00729 V=30.0 PL=1
MOVL C00730 V=130.0 PL=1
MOVL C00731 V=30.0 PL=1
MOVL C00732 V=130.0 PL=1
MOVL C00733 V=20.0 PL=1
MOVL C00734 V=130.0 PL=1
MOVL C00735 V=130.0 PL=1
MOVL C00736 V=30.0 PL=1
MOVL C00737 V=130.0 PL=1
MOVL C00738 V=60.0 PL=1
MOVL C00739 V=60.0 PL=1
MOVL C00740 V=60.0 PL=1
MOVL C00741 V=60.0 PL=1
MOVL C00742 V=130.0 PL=1
MOVL C00743 V=30.0 PL=1
MOVL C00744 V=30.0 PL=1
MOVL C00745 V=30.0 PL=1
MOVL C00746 V=30.0 PL=1
MOVL C00747 V=30.0 PL=1
MOVL C00748 V=30.0 PL=1
MOVL C00749 V=30.0 PL=1
MOVL C00750 V=30.0 PL=1
MOVL C00751 V=130.0 PL=1
MOVL C00752 V=130.0 PL=1
MOVL C00753 V=30.0 PL=1
MOVL C00754 V=130.0 PL=1
MOVL C00755 V=30.0 PL=1
MOVL C00756 V=130.0 PL=1
MOVL C00757 V=30.0 PL=1
MOVL C00758 V=130.0 PL=1
MOVL C00759 V=20.0 PL=1
MOVL C00760 V=130.0 PL=1
MOVL C00761 V=130.0 PL=1
MOVL C00762 V=30.0 PL=1
MOVL C00763 V=130.0 PL=1
MOVL C00764 V=60.0 PL=1
MOVL C00765 V=60.0 PL=1
MOVL C00766 V=60.0 PL=1
MOVL C00767 V=60.0 PL=1
MOVL C00768 V=130.0 PL=1
MOVL C00769 V=30.0 PL=1
MOVL C00770 V=30.0 PL=1
MOVL C00771 V=30.0 PL=1
MOVL C00772 V=30.0 PL=1
MOVL C00773 V=30.0 PL=1
MOVL C00774 V=30.0 PL=1
MOVL C00775 V=30.0 PL=1
MOVL C00776 V=30.0 PL=1
MOVL C00777 V=130.0 PL=1
MOVL C00778 V=130.0 PL=1
MOVL C00779 V=30.0 PL=1
MOVL C00780 V=130.0 PL=1
MOVL C00781 V=30.0 PL=1
MOVL C00782 V=130.0 PL=1
MOVL C00783 V=30.0 PL=1
MOVL C00784 V=130.0 PL=1
MOVL C00785 V=20.0 PL=1
MOVL C00786 V=130.0 PL=1
MOVL C00787 V=130.0 PL=1
MOVL C00788 V=30.0 PL=1
MOVL C00789 V=130.0 PL=1
MOVL C00790 V=60.0 PL=1
MOVL C00791 V=60.0 PL=1
MOVL C00792 V=60.0 PL=1
MOVL C00793 V=60.0 PL=1
MOVL C00794 V=130.0 PL=1
MOVL C00795 V=30.0 PL=1
MOVL C00796 V=30.0 PL=1
MOVL C00797 V=30.0 PL=1
MOVL C00798 V=30.0 PL=1
MOVL C00799 V=30.0 PL=1
MOVL C00800 V=30.0 PL=1
MOVL C00801 V=30.0 PL=1
MOVL C00802 V=30.0 PL=1
MOVL C00803 V=130.0 PL=1
MOVL C00804 V=130.0 PL=1
MOVL C00805 V=30.0 PL=1
MOVL C00806 V=130.0 PL=1
MOVL C00807 V=30.0 PL=1
MOVL C00808 V=130.0 PL=1
MOVL C00809 V=30.0 PL=1
MOVL C00810 V=130.0 PL=1
MOVL C00811 V=20.0 PL=1
MOVL C00812 V=130.0 PL=1
MOVL C00813 V=130.0 PL=1
MOVL C00814 V=30.0 PL=1
MOVL C00815 V=130.0 PL=1
MOVL C00816 V=60.0 PL=1
MOVL C00817 V=60.0 PL=1
MOVL C00818 V=60.0 PL=1
MOVL C00819 V=60.0 PL=1
MOVL C00820 V=130.0 PL=1
MOVL C00821 V=30.0 PL=1
MOVL C00822 V=30.0 PL=1
MOVL C00823 V=30.0 PL=1
MOVL C00824 V=30.0 PL=1
MOVL C00825 V=30.0 PL=1
MOVL C00826 V=30.0 PL=1
MOVL C00827 V=30.0 PL=1
MOVL C00828 V=30.0 PL=1
MOVL C00829 V=130.0 PL=1
MOVL C00830 V=130.0 PL=1
MOVL C00831 V=30.0 PL=1
MOVL C00832 V=130.0 PL=1
MOVL C00833 V=30.0 PL=1
MOVL C00834 V=130.0 PL=1
MOVL C00835 V=30.0 PL=1
MOVL C00836 V=130.0 PL=1
MOVL C00837 V=20.0 PL=1
MOVL C00838 V=130.0 PL=1
MOVL C00839 V=130.0 PL=1
MOVL C00840 V=30.0 PL=1
MOVL C00841 V=130.0 PL=1
MOVL C00842 V=60.0 PL=1
MOVL C00843 V=60.0 PL=1
MOVL C00844 V=60.0 PL=1
MOVL C00845 V=60.0 PL=1
MOVL C00846 V=130.0 PL=1
MOVL C00847 V=30.0 PL=1
MOVL C00848 V=30.0 PL=1
MOVL C00849 V=30.0 PL=1
MOVL C00850 V=30.0 PL=1
MOVL C00851 V=30.0 PL=1
MOVL C00852 V=30.0 PL=1
MOVL C00853 V=30.0 PL=1
MOVL C00854 V=30.0 PL=1
MOVL C00855 V=130.0 PL=1
MOVL C00856 V=130.0 PL=1
MOVL C00857 V=30.0 PL=1
MOVL C00858 V=130.0 PL=1
MOVL C00859 V=30.0 PL=1
MOVL C00860 V=130.0 PL=1
MOVL C00861 V=30.0 PL=1
MOVL C00862 V=130.0 PL=1
MOVL C00863 V=20.0 PL=1
MOVL C00864 V=130.0 PL=1
MOVL C00865 V=130.0 PL=1
MOVL C00866 V=30.0 PL=1
MOVL C00867 V=130.0 PL=1
MOVL C00868 V=60.0 PL=1
MOVL C00869 V=60.0 PL=1
MOVL C00870 V=60.0 PL=1
MOVL C00871 V=60.0 PL=1
MOVL C00872 V=130.0 PL=1
MOVL C00873 V=30.0 PL=1
MOVL C00874 V=30.0 PL=1
MOVL C00875 V=30.0 PL=1
MOVL C00876 V=30.0 PL=1
MOVL C00877 V=30.0 PL=1
MOVL C00878 V=30.0 PL=1
MOVL C00879 V=30.0 PL=1
MOVL C00880 V=30.0 PL=1
MOVL C00881 V=130.0 PL=1
MOVL C00882 V=130.0 PL=1
MOVL C00883 V=30.0 PL=1
MOVL C00884 V=130.0 PL=1
MOVL C00885 V=30.0 PL=1
MOVL C00886 V=130.0 PL=1
MOVL C00887 V=30.0 PL=1
MOVL C00888 V=130.0 PL=1
MOVL C00889 V=20.0 PL=1
MOVL C00890 V=130.0 PL=1
MOVL C00891 V=130.0 PL=1
MOVL C00892 V=30.0 PL=1
MOVL C00893 V=130.0 PL=1
MOVL C00894 V=60.0 PL=1
MOVL C00895 V=60.0 PL=1
MOVL C00896 V=60.0 PL=1
MOVL C00897 V=60.0 PL=1
MOVL C00898 V=130.0 PL=1
MOVL C00899 V=30.0 PL=1
MOVL C00900 V=30.0 PL=1
MOVL C00901 V=30.0 PL=1
MOVL C00902 V=30.0 PL=1
MOVL C00903 V=30.0 PL=1
MOVL C00904 V=30.0 PL=1
MOVL C00905 V=30.0 PL=1
MOVL C00906 V=30.0 PL=1
MOVL C00907 V=130.0 PL=1
MOVL C00908 V=130.0 PL=1
MOVL C00909 V=30.0 PL=1
MOVL C00910 V=130.0 PL=1
MOVL C00911 V=30.0 PL=1
MOVL C00912 V=130.0 PL=1
MOVL C00913 V=30.0 PL=1
MOVL C00914 V=130.0 PL=1
MOVL C00915 V=20.0 PL=1
MOVL C00916 V=130.0 PL=1
MOVL C00917 V=130.0 PL=1
MOVL C00918 V=30.0 PL=1
MOVL C00919 V=130.0 PL=1
MOVL C00920 V=60.0 PL=1
MOVL C00921 V=60.0 PL=1
MOVL C00922 V=60.0 PL=1
MOVL C00923 V=60.0 PL=1
MOVL C00924 V=130.0 PL=1
MOVL C00925 V=30.0 PL=1
MOVL C00926 V=30.0 PL=1
MOVL C00927 V=30.0 PL=1
MOVL C00928 V=30.0 PL=1
MOVL C00929 V=30.0 PL=1
MOVL C00930 V=30.0 PL=1
MOVL C00931 V=30.0 PL=1
MOVL C00932 V=30.0 PL=1
MOVL C00933 V=130.0 PL=1
MOVL C00934 V=130.0 PL=1
MOVL C00935 V=30.0 PL=1
MOVL C00936 V=130.0 PL=1
MOVL C00937 V=30.0 PL=1
MOVL C00938 V=130.0 PL=1
MOVL C00939 V=30.0 PL=1
MOVL C00940 V=130.0 PL=1
MOVL C00941 V=20.0 PL=1
MOVL C00942 V=130.0 PL=1
MOVL C00943 V=130.0 PL=1
END
